	        IF (#new_packet) THEN
	            #_State := #STATE_INIT;
	        END_IF;
	        
	        
	END_CASE;
	
	EndAutomat:
	
	#CMD_CloseLodems := NOT #CMD_OpenLodems;
	
	// make new layer
	// 
	#make_gasket_layer := #s_lay_cmd_permission AND NOT #gaskets_busy AND (NOT (#mode_no_gasket OR #last_lay));
	
	
	
END_FUNCTION_BLOCK

FUNCTION "BoardDefinePosition" : Int
{ S7_Optimized_Access := 'FALSE' }
AUTHOR : Aspir
VERSION : 0.1
   VAR_INPUT 
      EnableRolling : Bool;   // нужна ли раскатка пакета
      PackL : Int;   // длина пакета с раскаткой
      PlankL : Int;   // длина доски
   END_VAR

   VAR CONSTANT 
      SafetyOffset : Int := 100;
   END_VAR


BEGIN
	IF (#EnableRolling) THEN
	    #BoardDefinePosition := #PackL;
	ELSIF (#PlankL = 0) THEN
	    #BoardDefinePosition := 6000;
	ELSE
	    #BoardDefinePosition := #PlankL + #SafetyOffset;
	END_IF;
END_FUNCTION

FUNCTION "SolveMovBoardPos" : Int
{ S7_Optimized_Access := 'FALSE' }
VERSION : 0.1
   VAR_INPUT 
      PlankLength : Int;
      Max_pos : Int;
      Min_pos : Int;
      Offset_chess : Int;
      PulseCount : Int;
   END_VAR

   VAR_TEMP 
      PlankLength_tmp : Int;
      Sub : Int;
      k : Real;
      b : Real;
   END_VAR


BEGIN
	IF (#PlankLength > #Max_pos) THEN
	    #PlankLength_tmp := #Max_pos;
	ELSIF (#PlankLength < #Min_pos) THEN
	    #PlankLength_tmp := #Min_pos;
	ELSE
	    #PlankLength_tmp := #PlankLength;
	END_IF;
	
	#Sub := (#Min_pos - #Max_pos);
	
	#k := INT_TO_REAL(#PulseCount) / #Sub;
	
	#b := - #Max_pos * #k;
	
	#SolveMovBoardPos := TRUNC_INT((#PlankLength_tmp + #Offset_chess)*#k + #b);
END_FUNCTION

FUNCTION_BLOCK "MovableBoard_CTRL"
{ S7_Optimized_Access := 'FALSE' }
VERSION : 0.1
   VAR_INPUT 
      BoardBase : Bool;   //   сигнал с дальнего концевика борта (знаем его позицию точно)
      ModeChanged : Bool;   //  был изменен режим
      Reset : Bool;   //   сбросить базу и позицию
      EncPos : Byte;   //   показания энкодера (код Грея)
      SetPos : Int;   //   абсолютное положение борта в импульсах
   END_VAR

   VAR_OUTPUT 
      CMD_Fwd : Bool;   //   команда на движение вперед
      CMD_Bwd : Bool;   //   команда на движение назад
      CMD_UP : Bool;   //   команда опустить борт
      CMD_DOWN : Bool;   //   команда поднять борт
      AutoMode : Bool;
      ResetVirtualPos : Bool;
      Position : Int;
   END_VAR

   VAR 
      DefinitionTag : Bool;   //   была определена позиция (база борта)
      ChangingPos : Bool;   //  в состоянии изменения позиции
      ShutUpAuto : Bool;   //  позицию изменил
      startOffset : Int;   //  начальный сдвиг
      curMicroPos : Int;
      curMicroPos_old : Int;
      curMacroPos : Int;
   END_VAR


BEGIN
	#ResetVirtualPos := FALSE;
	
	// условия для учета "перескоков" абсолютного энкодера на 256 позиций
	#curMicroPos := "Rev_G"(#EncPos);
	IF (#curMicroPos_old - #curMicroPos > 200) THEN
	    #curMacroPos := #curMacroPos + 1;
	END_IF;
	IF (#curMicroPos - #curMicroPos_old > 200) THEN
	    #curMacroPos := #curMacroPos - 1;
	END_IF;
	
	
	// Итоговое положение
	#Position := 256 * #curMacroPos + #curMicroPos - #startOffset;
	
	// Сброс базы
	IF #Reset THEN
	    #DefinitionTag := False;
	    #ChangingPos := FALSE;
	    #CMD_UP := FALSE;
	    #CMD_DOWN := FALSE;
	    
	    #ResetVirtualPos := TRUE;
	END_IF;
	
	// Доведем борт до концевика для уверенности в базе (нулевой точке)
	IF NOT #DefinitionTag THEN
	    #AutoMode := TRUE;
	    #CMD_UP := TRUE;
	    #CMD_DOWN := FALSE;
	    #CMD_Fwd := TRUE;
	    #CMD_Bwd := FALSE;
	    // Если дошли до дальнего концевика, знаем где мы, обнулим счетчик оборотов
	    IF (#BoardBase) THEN
	        #DefinitionTag := TRUE;
	        #ShutUpAuto := TRUE;
	        #curMacroPos := 0;
	        #startOffset := #curMicroPos;
	    END_IF;
	END_IF;
	
	
	IF (#ShutUpAuto) THEN
	    #AutoMode := False;
	    #ShutUpAuto := FALSE;
	END_IF;
	
	
	#ChangingPos := (#ChangingPos OR #ModeChanged);
	
	IF #ChangingPos AND #DefinitionTag THEN
	    #AutoMode := True;
	    #CMD_UP := True;
	    #CMD_DOWN := False;
	    
	    IF (ABS_INT(#Position - #SetPos) < 12) THEN
	        #ChangingPos := FALSE;
	        #ShutUpAuto := TRUE;
	        #CMD_UP := #SetPos < 30;
	        #CMD_DOWN := NOT #CMD_UP;
	        #CMD_Bwd := FALSE;
	        #CMD_Fwd := FALSE;
	        
	    ELSIF #Position > #SetPos THEN
	        #CMD_Bwd := FALSE;
	        #CMD_Fwd := TRUE;
	        
	    ELSE
	        #CMD_Bwd := TRUE;
	        #CMD_Fwd := FALSE;
	    END_IF;
	END_IF;
	
	
	#curMicroPos_old := #curMicroPos;
END_FUNCTION_BLOCK

FUNCTION "Rev_G" : Int
{ S7_Optimized_Access := 'FALSE' }
VERSION : 0.1
   VAR_INPUT 
      g_code : Byte;   // число (Код Грея)
   END_VAR

   VAR_TEMP 
      n : Byte;
   END_VAR


BEGIN
	#n := 0;
	
	WHILE NOT (#g_code = 0) DO
	    // Statement section WHILE
	    #n := #n XOR #g_code;
	    #g_code := SHR(IN := #g_code, N := 1);
	END_WHILE;
	
	#Rev_G := BYTE_TO_INT(#n);
END_FUNCTION

FUNCTION_BLOCK "FB_IM_PFM"
{ S7_Optimized_Access := 'FALSE' }
VERSION : 0.1
   VAR 
      M_233_Fork_PFM { S7_SetPoint := 'False'} : "FB_IM2x4";   // Вилы основной ПФМ
      M_232_Elevator_PFM : "FB_IM2x2S";   // Лифт основной ПФМ
      M_317_Carousel : "drive_CB_2x1";
      Elevator_brake_timer {InstructionName := 'TON'; LibVersion := '1.0'} : TON;
   END_VAR

   VAR_TEMP 
      Sert : Word;
   END_VAR


BEGIN
	
	REGION M_233
	    // Statement section REGION
	    #M_233_Fork_PFM(OnSig:="DGI".S15_2,
	                    OnSigLow:="DGI".S15_1,
	                    OffSig:= "DGI".S14_7,
	                    OffSigLow:="DGI".S15_0,
	                    sigFeedback:="DGI".F233K1 AND "DGI".K1_233U1,
	                    hasFeedback:=TRUE,
	                    Ready:="ALG".Ready_Sorting,
	                    Reset:="ALG".Reset OR "DGI".S76_2,
	                    btnAU:="ALG".Auto_Sorting OR "ServDB".M_233.BtnAU,
	                    btnDU:= NOT "ALG".Auto_Sorting AND "ServDB".M_233.BtnDU,
	                    prmDU:=TRUE,
	                    btnDU_ON:="ServDB".M_233.BtnFwd,
	                    btnDU_OF:= "ServDB".M_233.BtnBwd,
	                    btnDUStop:="ServDB".M_233.BtnCmdStop,
	                    btnMU:=NOT ("ALG".Auto_Sorting OR "ServDB".M_233.BtnDU),
	                    btnMU_ON:="DGI".S78_0,
	                    btnMU_OF:="DGI".E78_1,
	                    protection:=false,
	                    Set_T_notON:=T#20s,
	                    Set_T_notOFF:=T#20s,
	                    Set_T_notCMD:=T#500ms,
	                    Set_T_notFeedBack:=T#500ms,
	                    SpeedOn:=20,
	                    SpeedOnLow:=10,
	                    SpeedOff:=20,
	                    SpeedOffLow:=10,
	                    SpeedDU:="ServDB".M_233.SetSpeedDU,
	                    AU=>"ServDB".M_233.AU,
	                    DU=>"ServDB".M_233.DU,
	                    MU=>"ServDB".M_233.MU,
	                    Fault=>"ServDB".M_233.Fault,
	                    onOutFWD=>"ServDB".M_233.CMD_ON,
	                    onOutBWD=>"ServDB".M_233.CMD_OFF,
	                    PRM_btnDU_ON=>"ServDB".M_233.PrmBtnDU_ON,
	                    PRM_btnDU_OFF=>"ServDB".M_233.PrmBtnDU_OF
	                   
	    );
	    
	    
	    "K1-233X1" := "ALG".Ready_Sorting;
	    "K1-233U2" := #M_233_Fork_PFM.onOutFWD OR #M_233_Fork_PFM.onOutBWD;
	    "K1-233U2.2" := #M_233_Fork_PFM.onOutFWD;
	END_REGION
	
	REGION M_232
	    // Statement section REGION
	    #M_232_Elevator_PFM(onSig := "DGI".S16_2,
	                        offSig := "DGI".S16_1,
	                        sigFeedback := "DGI".F232K1 AND "DGI".K1_215U1,
	                        hasFeedback := true,
	                        btnUp := "ServDB".M_232.BtnFwd,
	                        btnDown := "ServDB".M_232.BtnBwd,
	                        btnStop := "ServDB".M_232.BtnCmdStop,
	                        Ready := "ALG".Ready_Sorting,
	                        Reset := "ALG".Reset OR "DGI".S76_2,
	                        prmDU := true,
	                        btnAU := "ServDB".M_232.BtnAU OR "ALG".Auto_Sorting,
	                        btnDU := "ServDB".M_232.BtnDU,
	                        btnMU := "DGI".E86_1 OR "DGI".E78_5 OR "DGI".S86_0 OR "DGI".S78_4 OR NOT ("ALG".Auto_Sorting OR "ServDB".M_232.BtnDU),
	                        btnMU_ON := "DGI".E86_1 OR "DGI".E78_5,
	                        btnMU_OF := "DGI".S86_0 OR "DGI".S78_4,
	                        set_time_notOn := T#1500ms,
	                        set_time_notOff := T#5000ms,
	                        set_time_notCMD := T#2000ms,
	                        setSpeedDU := "ServDB".M_232.SetSpeedDU,
	                        AU => "ServDB".M_232.AU,
	                        DU => "ServDB".M_232.DU,
	                        MU => "ServDB".M_232.MU,
	                        Fault => "ServDB".M_232.Fault,
	                        outFWD => "ServDB".M_232.CMD_ON,
	                        outBKD => "ServDB".M_232.CMD_OFF,
	                        setSpeed => "ServDB".M_317.SetSpeed
	    );
	    
	    "K1-232X1" := "ALG".Ready_Sorting;
	    // Управление тормозом
	    #Elevator_brake_timer(IN := #M_232_Elevator_PFM.outFWD XOR #M_232_Elevator_PFM.outBKD,
	                          PT := T#50ms
	    );
	    
	    "K1-232X1.1" := #Elevator_brake_timer.Q AND "DGI".K1_215U1;
	    
	    "K1-215U2.2" := #M_232_Elevator_PFM.outBKD;
	    "K1-215U2" := #M_232_Elevator_PFM.outFWD OR #M_232_Elevator_PFM.outBKD;
	END_REGION
	
	REGION M_317
	    
	    (* #M_317_Gasket_Carousel(OnSig:="DGI".F317K1 AND "DGI".K1_317U1,
	                           OnCom:= ("FB_Gasket_Carousel_DB".Carousel_FWD AND (NOT "B18.0")) OR "FB_Gasket_Carousel_DB".Carousel_BWD,
	                           Ready:="ALG".Ready_Sorting,
	                           Reset:="DGI".S76_2 OR "ALG".Reset,
	                           btnAU:= "ServDB".M_317.BtnAU OR "ALG".Auto_Sorting,
	                           btnDU:="ServDB".M_317.BtnDU,
	                           prmDU:=true,
	                           btnDU_ON:="ServDB".M_317.BtnFwd OR "ServDB".M_317.BtnBwd,
	                           btnDU_OF:= "ServDB".M_317.BtnCmdStop,
	                           btnMU:=NOT ("ServDB".M_317.BtnDU OR "ALG".Auto_Sorting) OR ("FB_Gasket_Carousel_DB".s_man_cntl AND "ALG".Auto_Sorting),
	                           btnMU_ON:="DGI".S84_1 OR "DGI".E84_2,
	                           btnMU_OF:= NOT ("DGI".S84_1 OR "DGI".E84_2),
	                           btn_Back_ON:= "ServDB".M_317.BtnBwd OR "DGI".E84_2 OR "FB_Gasket_Carousel_DB".Carousel_BWD,
	                           btn_Back_OFF:= NOT ("ServDB".M_317.BtnBwd OR "DGI".E84_2 OR "FB_Gasket_Carousel_DB".Carousel_BWD),
	                           Set_T_notON:=T#500ms,
	                           Set_T_notOFF:=T#500ms,
	                           setSpeedDU:="ServDB".M_317.SetSpeedDU,
	                           AU=>"ServDB".M_317.AU,
	                           DU=>"ServDB".M_317.DU,
	                           MU=>"ServDB".M_317.MU,
	                           BACK=>"ServDB".M_317.BACK,
	                           Alarm=>"ServDB".M_317.Alarm,
	                           Fault=>"ServDB".M_317.Fault,
	                           onOutFWD=>"ServDB".M_317.CMD_ON,
	                           onOutBWD=>"ServDB".M_317.CMD_OFF,
	                           PRM_btnDU_ON=>"ServDB".M_317.PrmBtnDU_ON,
	                           PRM_btnDU_OFF=>"ServDB".M_317.PrmBtnDU_OF,
	                           PRMbtn_Back_ON=>"ServDB".M_317.PRMbtn_Back_ON,
	                           PRMbtn_Back_OFF=>"ServDB".M_317.PRMbtn_Back_OFF,
	                           setSpeed=>"ServDB".M_317.SetSpeed
	    );
	    
	    
	    "K1-317X1" := "ALG".Ready_Sorting;
	    "K1-317U2" := #M_317_Gasket_Carousel.onOutFWD OR #M_317_Gasket_Carousel.onOutBWD;
	    "K1-317X1.1" := #M_317_Gasket_Carousel.onOutFWD OR #M_317_Gasket_Carousel.onOutBWD;
	    "K1-317U2.2" := #M_317_Gasket_Carousel.onOutBWD;
	    
	    *)
	    
	    #M_317_Carousel(i_ready := "ALG".Ready_Sorting,
	                    i_feedback := "DGI".F317K1 AND "DGI".K1_317U1,
	                    i_reset := "DGI".S76_2 OR "ALG".Reset,
	                    i_au_req := "ALG".Auto_Sorting,
	                    cmd_fwd := "FB_Gasket_Carousel_DB".Carousel_FWD AND NOT "B18.0",
	                    cmd_bwd := "FB_Gasket_Carousel_DB".Carousel_BWD,
	                    i_mu_req := ("FB_Gasket_Carousel_DB".s_man_cntl AND "ALG".Auto_Sorting) OR NOT ("ALG".Auto_Sorting OR "ServDB".M_317.BtnDU),
	                    mu_fwd := "DGI".S84_1,
	                    mu_bwd := "DGI".E84_2,
	                    i_du_req := "ServDB".M_317.BtnDU,
	                    du_fwd := "ServDB".M_317.BtnFwd,
	                    du_bwd := "ServDB".M_317.BtnBwd,
	                    i_speed_au := "FB_Gasket_Carousel_DB".Carousel_Speed,
	                    i_speed_mu_du := 7.0,
	                    ////////////////////////////////
	                    o_au => "ServDB".M_317.AU,
	                    o_du => "ServDB".M_317.DU,
	                    o_mu => "ServDB".M_317.MU,
	                    alarm => "ServDB".M_317.Alarm,
	                    o_fwd => "ServDB".M_317.CMD_ON,
	                    o_bwd => "ServDB".M_317.CMD_OFF);
	    
	    "K1-317X1" := "ALG".Ready_Sorting;
	    "K1-317U2" := #M_317_Carousel.o_fwd OR #M_317_Carousel.o_bwd;
	    "K1-317X1.1" := #M_317_Carousel.o_brake;
	    "K1-317U2.2" := #M_317_Carousel.o_bwd;
	    
	    #Sert := UNSCALE(IN := #M_317_Carousel.o_speed_vfd, HI_LIM := 50.0, LO_LIM := -50.0, BIPOLAR := TRUE, OUT => "K1-317U":P);
	    
	    
	    
	    
	END_REGION
END_FUNCTION_BLOCK

FUNCTION_BLOCK "FB_IM2x4"
{ S7_Optimized_Access := 'FALSE' }
AUTHOR : Ivanez
VERSION : 0.1
//Исполнительный механизм (2 команды, 4 положения - 2 конечных, 2 замедление)
   VAR_INPUT 
      OnSig : Bool;   //      Сигнал сработавшего открытого (выдвинутого)
      OnSigLow : Bool;   //      Сигнал сработавшего открытого (выдвинутого) замедление
      OffSig : Bool;   //      Сигнал сработавшего закрытого (задвинутого)
      OffSigLow : Bool;   //      Сигнал сработавшего закрытого (задвинутого) замедление
      OnCom : Bool;   //      Команда включения в автоматическом режиме
      OffCom : Bool;   //      Команда отключения в автоматическом режиме
      sigFeedback : Bool;   //      Обратная связь о том что устройство передвигается
      hasFeedback : Bool;   //      Флаг о наличии обратной связи по движению
      Ready : Bool;   //      Условие готовности
      Reset : Bool;   //      Сброс
      btnAU : Bool;   //      Перевести в Автоматическое управление
      btnDU : Bool;   //      Перевести в Дистанционное управление
      prmDU : Bool;   //      Разрешение на перевод в ДУ
      btnDU_ON : Bool;   //      Выдвинуть в дистанционном управлении
      btnDU_OF : Bool;   //      Задвинуть в дистанционном управлении
      btnDUStop : Bool;   //      Кнопка Останов
      btnMU : Bool;   //      Перевести в местное управление
      btnMU_ON : Bool;   //      Включить в местном управлении
      btnMU_OF : Bool;   //      Отключить в местном управлении
      protection : Bool;   //      Условие включение защиты
      Set_T_notON : Time;   //      Задержа на формирование неоткрытия
      Set_T_notOFF : Time;   //      Задержа на формирование незакрытия
      Set_T_notCMD : Time;   //      Задержа на формирование отсутсвия команды
      Set_T_notFeedBack : Time;   // Задержка на формирование ошибки отсутствия обратной связи
      SpeedOn : Real;   //     Задание на скорость выдвижения
      SpeedOnLow : Real;   //     Задание на скорость выдвижения низкая
      SpeedOff : Real;   //     Задание на скорость задвижения
      SpeedOffLow : Real;   //     Задание на скорость задвижения низкая
      SpeedDU : Real;   //     Задание на скорость в ДУ
   END_VAR

   VAR_OUTPUT 
      AU : Bool;   //      Автоматическое управление (АУ)
      DU : Bool;   //      Дистанционное управление (ДУ)
      MU : Bool;   //      Местное управление (МУ)
      notON : Bool;   //      Предупреждение о невключении
      notOFF : Bool;   //      Предупреждение о неотключении
      notCMD : Bool;   //      Предупреждение об отсутствие команды
      notFeedBack : Bool;   // Предупреждение об отсутствии обратной связи
      Fault : Bool;   //      Неисправность
      onOutFWD : Bool;   //      Сигнал на открытие (выдвинуть)
      onOutBWD : Bool;   //      Сигнал на закрытие (задвинуть)
      PRM_btnDU_ON : Bool;   //      Разрешение кнопки включения в ДУ
      PRM_btnDU_OFF : Bool;   //      Разрешение кнопки отключения в ДУ
      SetSpeed : Real;   //     Задание на ПЧ
   END_VAR

   VAR 
      speedLow_forward : Bool;
      speedLow_revers : Bool;
      checker_forward : Bool;
      checker_revers : Bool;
      unkn_state : Bool;   //     Неизвестное состояние
      wrong_state : Bool;   //     Некорректное состояние
      sigOnOut : Bool;   //      Сигналоткрытия
      sigOffOut : Bool;   //      Сигнал закрытия
      T_notON_TON {InstructionName := 'TON'; LibVersion := '1.0'; S7_SetPoint := 'False'} : TON;   //      Таймер неоткрытия
      T_notOFF_TON {InstructionName := 'TON'; LibVersion := '1.0'; S7_SetPoint := 'False'} : TON;   //      Таймер незакрытия
      T_notCMD_TON {InstructionName := 'TON'; LibVersion := '1.0'; S7_SetPoint := 'False'} : TON;   //      Таймер отстутствия
      T_notFeedBack_TON {InstructionName := 'TON'; LibVersion := '1.0'} : TON;   // Таймер отсутствия обратной связи
   END_VAR


BEGIN
	
	//Формирование автоматического управления
	IF #btnAU THEN
	    #AU := true;
	    #DU := false;
	    #MU := false;
	END_IF;
	//Формирование дистанционного управления 
	IF #btnDU THEN
	    #DU := true;
	    #AU := false;
	    #MU := false;
	END_IF;
	//Формирование местного управления
	IF #btnMU THEN
	    #MU := true;
	    #AU := false;
	    #DU := false;
	END_IF;
	
	IF NOT #AU AND NOT #DU AND NOT #MU THEN
	    #MU := true;
	END_IF;
	
	//Разрешения кнопок управления
	#PRM_btnDU_ON := (NOT #OnSig AND #DU OR #notON);
	#PRM_btnDU_OFF := (NOT #OffSig AND #DU OR #notOFF);
	
	
	// Контроль скорости
	// 
	// триггеры замедления
	// 
	#speedLow_forward := (#speedLow_forward OR #OnSigLow AND #sigOnOut) AND NOT (#OnSig OR #OnSigLow AND #sigOffOut);
	#speedLow_revers := (#speedLow_revers OR #OffSigLow AND #sigOffOut) AND NOT (#OffSig OR #OffSigLow AND #sigOnOut);
	#checker_forward := (#checker_forward OR #OffSig) AND NOT #OffSigLow;
	#checker_revers := (#checker_revers OR #OnSig) AND NOT #OnSigLow;
	
	IF (#sigOnOut) THEN
	    IF (#speedLow_forward OR #checker_revers) THEN
	        #SetSpeed := #SpeedOnLow;
	    ELSE
	        #SetSpeed := #SpeedOn;
	    END_IF;
	    
	    
	ELSIF (#sigOffOut) THEN
	    IF (#speedLow_revers OR #checker_forward) THEN
	        #SetSpeed := #SpeedOffLow;
	    ELSE
	        #SetSpeed := #SpeedOff;
	    END_IF;
	ELSE
	    #SetSpeed := 0;
	END_IF;
	
	//------------------------------------------------
	//Формирование выходного сигнала открытия (выдвижение)
	#sigOnOut := #Ready AND ((#sigOnOut
	OR #AU AND #OnCom
	OR #DU AND #btnDU_ON
	OR #MU AND #btnMU_ON)
	AND NOT (#OnSig
	OR #AU AND ( #OffCom)
	OR #DU AND (#btnDU_OF OR #btnDUStop)
	OR #MU AND (NOT #btnMU_ON OR #btnMU_OF)
	OR #notON
	OR #wrong_state
	));
	
	//Формирование выходного сигнала закрытия (задвижение)
	#sigOffOut := #Ready AND ((#sigOffOut
	OR #AU AND #OffCom
	OR #DU AND #btnDU_OF
	OR #MU AND #btnMU_OF)
	AND NOT (#OffSig
	OR #AU AND (#OnCom)
	OR #DU AND (#btnDU_ON OR #btnDUStop)
	OR #MU AND (#btnMU_ON OR NOT #btnMU_OF)
	OR #notOFF
	OR #wrong_state
	));
	
	//Выбор выхода 
	#onOutFWD := #sigOnOut;
	#onOutBWD := #sigOffOut;
	
	
	//Неизвестное состояние
	#unkn_state := NOT (#OnSig OR #OffSig OR #onOutBWD OR #onOutFWD) AND NOT #Reset;
	
	//Некорректное состояние
	#wrong_state := (#wrong_state
	OR #OnSig AND #OffSig
	OR #OnSig AND #OffSigLow
	OR #OnSigLow AND #OffSigLow
	OR #OnSigLow AND #OffSig
	) AND NOT #Reset;
	
	
	#T_notON_TON(
	             IN := ( #sigOnOut AND NOT #sigOffOut AND NOT #OnSig AND NOT #Reset ),
	             PT := #Set_T_notON
	);
	
	#notON := (#notON OR #T_notON_TON.Q) AND NOT #Reset;
	
	#T_notCMD_TON(
	              IN := ( NOT #sigOnOut AND NOT #sigOffOut AND (#sigFeedback AND #hasFeedback) AND NOT #Reset),
	              PT := #Set_T_notCMD
	);
	
	#notCMD := (#notCMD OR #T_notCMD_TON.Q) AND NOT #Reset;
	
	
	#T_notOFF_TON(
	              IN := (NOT #sigOnOut AND #sigOffOut AND NOT #OffSig AND NOT #Reset),
	              PT := #Set_T_notOFF
	);
	
	#notOFF := (#notOFF OR #T_notOFF_TON.Q) AND NOT #Reset;
	
	#T_notFeedBack_TON(
	                   IN := (#sigOnOut OR #sigOffOut) AND NOT (#sigFeedback AND #hasFeedback) AND NOT #Reset,
	                   PT := #Set_T_notFeedBack
	);
	
	#notFeedBack := (#notFeedBack OR #T_notFeedBack_TON.Q) AND NOT #Reset;
	
	//Обобщенная неисправность
	#Fault := #notON OR #notOFF OR #notCMD OR #notFeedBack OR #wrong_state OR #unkn_state;
END_FUNCTION_BLOCK

FUNCTION_BLOCK "FB_IM2x2S"
{ S7_Optimized_Access := 'FALSE' }
VERSION : 0.1
//------------------------------------------------------------------------------------
//  Declaration of Variables
//------------------------------------------------------------------------------------
   VAR_INPUT 
      onSig : Bool;   //      Сигнал верхнего концевика
      offSig : Bool;   //      Сигнал нижнего концевика
      sigFeedback : Bool;   //      Обратная связь о том что устройство передвигается
      hasFeedback : Bool;   //      Флаг о наличии обратной связи по движению
      comUp : Bool;   //      Команда на подъем оборудования в автомате
      comDown : Bool;   //      Команда на спуск оборудования в автомате
      btnUp : Bool;   //      Кнопка на подъем лифта
      btnDown : Bool;   //      Кнопка на спуск лифта
      btnStop : Bool;   //      Кнопка Останов
      Ready : Bool;   //      Условие готовности
      Reset : Bool;   //      Сброс
      prmDU : Bool;   //      Разрешение на перевод в ДУ
      btnAU : Bool;   //      Команда на перевод в АУ
      btnDU : Bool;   //      Команда на пеервод в ДУ
      btnMU : Bool;
      btnMU_ON : Bool;   //      Включить в местном управлении
      btnMU_OF : Bool;   //      Отключить в местном управлении
      set_time_notOn : Time;   //      установка времени на неВКЛючение
      set_time_notOff : Time;   //      установка времени на неВЫКЛючение
      set_time_notCMD : Time;   //      установка времени отсутсивие команды
      setSpeedAU : Real;   //      Скорость в режиме автомат
      setSpeedDU : Real;   //      Скорость в режиме ДУoutputs
   END_VAR

   VAR_OUTPUT 
      AU : Bool;   //      Режим - Автомат
      DU : Bool;   //      Режим - ДистанционноеAlarm : Bool; // Авария
      MU : Bool;
      Fault : Bool;   //      Неисправность
      outFWD : Bool;   //      Сигнал о движении вверх (вперед)
      outBKD : Bool;   //      Сигнал о движении вниз (назад)
      notOn : Bool;   //      Сигнал на неВКЛючение
      notCMD : Bool;   //      Отсутствие команды
      notOff : Bool;   //      Сигнал на неВЫКЛючение
      wrong_state : Bool;   //      Некорректное состояние
      wrong_CMD : Bool;   // неверная команда
      setSpeed : Real;   //      скорость в автомате для частотникаvariables
   END_VAR

   VAR 
      timer_notOn {InstructionName := 'TON'; LibVersion := '1.0'} : TON;
      timer_notOff {InstructionName := 'TON'; LibVersion := '1.0'} : TON;
      timer_notCMD {InstructionName := 'TON'; LibVersion := '1.0'} : TON;
   END_VAR


BEGIN
	//Формирование автоматического управления
	IF #btnAU THEN
	    #AU := true;
	    #DU := false;
	    #MU := false;
	END_IF;
	//Формирование дистанционного управления 
	IF #btnDU THEN
	    #DU := true;
	    #AU := false;
	    #MU := false;
	END_IF;
	//Формирование местного управления
	IF #btnMU THEN
	    #MU := true;
	    #AU := false;
	    #DU := false;
	END_IF;
	
	IF NOT #AU AND NOT #DU AND NOT #MU THEN
	    #MU := true;
	END_IF;
	
	#outFWD := #Ready
	AND ((#outFWD
	OR #DU AND #btnUp
	OR #MU AND #btnMU_ON
	OR #AU AND #comUp)
	AND NOT (#Fault OR #onSig OR (#DU AND #btnStop) OR (#AU AND NOT #comUp) OR (#MU AND NOT #btnMU_ON))
	);
	
	#outBKD := #Ready
	AND ((#outBKD
	OR #DU AND #btnDown
	OR #MU AND #btnMU_OF
	OR #AU AND #comDown)
	AND NOT (#Fault OR #offSig OR (#DU AND #btnStop) OR (#AU AND NOT #comDown) OR (#MU AND NOT #btnMU_OF))
	);
	
	#timer_notOn(IN := (NOT #outBKD AND #outFWD) AND NOT (#sigFeedback AND #hasFeedback) AND NOT #Reset,
	             PT := #set_time_notOn);
	#notOn := (#notOn OR #timer_notOn.Q) AND NOT #Reset;
	
	// Не едет наверх
	// Проверка на отсутствие команд
	#timer_notCMD(IN := NOT (#outBKD OR #outFWD) AND (#sigFeedback AND #hasFeedback) AND NOT #Reset,
	              PT := #set_time_notCMD);
	#notCMD := (#notCMD OR #timer_notCMD.Q) AND NOT #Reset;
	
	// Не едет вниз
	#timer_notOff(IN := (#outBKD AND NOT #outFWD) AND NOT (#sigFeedback AND #hasFeedback) AND NOT #Reset,
	              PT := #set_time_notOff);
	#notOff := (#notOff OR #timer_notOff.Q) AND NOT #Reset;
	
	#wrong_CMD := (#wrong_CMD OR (#outFWD AND #outBKD)) AND NOT #Reset;
	
	#wrong_state := #onSig AND #offSig;
	
	#Fault := #notOn OR #notOff OR #notCMD OR #wrong_state OR #wrong_CMD;
	
	IF #DU THEN
	    #setSpeed := #setSpeedDU;
	ELSE
	    #setSpeed := #setSpeedAU;
	END_IF;
	
	
END_FUNCTION_BLOCK

FUNCTION_BLOCK "FB_HydroStations"
{ S7_Optimized_Access := 'FALSE' }
VERSION : 0.1
   VAR 
      Upor_resetter { S7_SetPoint := 'False'} : "CyclicSignal";
      Movable_side_resetter : "CyclicSignal";
      Gasket_Ramp_sync : "CyclicSignal";
      DefectDrop_resetter : "CyclicSignal";
      Board_Rotator { S7_SetPoint := 'False'} : "FB_IM2x0";   // переворот доски
      Defect_Drop : "FB_IM2x0";   // сброс в брак
      Upor_Sorting { S7_SetPoint := 'False'} : "FB_IM2x0";   // упор перед зоной оценки (поштучки)
      Upor_Defective : "FB_IM2x2";   // упоры ПФМ брака
      Gasket_Supplier { S7_SetPoint := 'False'} : "FB_IM2x0";   // выдача прокладки на карусель
      Gasket_Ramp : "FB_IM2x3";   // рама прокладок
      Gasket_Lodems : "FB_IM2x2";   // Стакан прокладок на раме
      Forks_Pitcher : "FB_IM2x2";   // подъемник вил ПФМ
      Movable_Side : "FB_IM2x0";   // Подвижный борт
      Upor_PFM : "FB_IM2x0";   // упоры перед пощштучной выдачей
      M_221_Large_HydroStationDrive : "FB_HySt_Drive_PassValve";   // двигатель маленькой гидростанции
      M_337_Small_HydroStationDrive : "FB_HySt_Drive_PassValve";   // двигатель большой гидростанции
   END_VAR


BEGIN
	REGION Small_HydroStationMechs
	    // Statement section REGION
	    
	    #Board_Rotator(Ready:="ALG".Ready_Sorting AND #M_337_Small_HydroStationDrive.CMD_DriveOn,
	                   Reset:="ALG".Reset,
	                   btnMU := TRUE,
	                   btnMU_On:="DGI".S88_7,
	                   btnMU_Off:=NOT "DGI".S88_7,
	                   set_T_On:=T#1s,
	                   set_T_Off:=T#1s,
	                   outFwd=> "Y223_1",
	                   outBwd=>"Y223_2"
	    );
	    
	    #DefectDrop_resetter(count:=240,
	                         Meandr_counter:="ALG".Meandr);
	    
	    #Defect_Drop(
	                 Ready:="ALG".Ready_Sorting AND #M_337_Small_HydroStationDrive.CMD_DriveOn,
	                 Reset:="ALG".Reset OR #DefectDrop_resetter.change,
	                 btnAU:= "ALG".Auto_Sorting,
	                 set_T_On:=T#2s,
	                 set_T_Off:=T#2200ms,
	                 outFwd => "Y223_4",
	                 outBwd => "Y223_3"
	    );
	    
	    #Upor_Sorting(Ready := "ALG".Ready_Sorting  AND #M_337_Small_HydroStationDrive.CMD_DriveOn,
	                  Reset := "ALG".Reset,
	                  btnAU := "ALG".Auto_Sorting,
	                  btnMU:=NOT ("ALG".Auto_Sorting),
	                  btnMU_On:= "DGI".S80_0,
	                  btnMU_Off:= "DGI".E80_1,
	                  set_T_On := T#1s,
	                  set_T_Off := T#500ms,
	                  outFwd => "Y323_2",
	                  outBwd => "Y323_1"
	    );
	    
	    #Upor_Defective(OnSig:="DGI".FC_23_6,
	                    OffSig:="DGI".FC_23_7,
	                    Ready:="ALG".Ready_defect AND #M_337_Small_HydroStationDrive.CMD_DriveOn,
	                    Reset:="ALG".Reset OR "DGI".S76_2,
	                    btnAU:="ALG".Auto_defect,
	                    btnMU:="DGI".S90_6 OR "DGI".E90_7, // OR "DGI".S80_0 OR "DGI".E80_1,
	                    btnMU_ON:= "DGI".S90_6,
	                    btnMU_OF:="DGI".E90_7,
	                    Set_T_notON:=T#7s,
	                    Set_T_notOFF:=T#7s,
	                    onOutFWD=>"Upor_brak_up",
	                    onOutBWD=>"Upor_brak_down"
	                    
	    );
	    
	END_REGION
	
	REGION Large_HydroStationMechs
	    // Statement section REGION
	    // 
	
	    #Gasket_Supplier(Ready := "ALG".Ready_Sorting AND #M_221_Large_HydroStationDrive.CMD_DriveOn,
	                     Reset := "ALG".Reset OR "DGI".S76_2,
	                     btnAU := "ALG".Auto_Sorting,
	                     btnDU:="ServDB".GasketSupplier.BtnDU,
	                     btnMU:=NOT ("ALG".Auto_Sorting OR "ServDB".GasketSupplier.BtnDU),
	                     btnDU_On:="ServDB".GasketSupplier.BtnFwd,
	                     btnDU_Off:="ServDB".GasketSupplier.BtnBwd,
	                     set_T_On := T#1s,
	                     set_T_Off := T#700ms,
	                     AU=>"ServDB".GasketSupplier.AU,
	                     DU=>"ServDB".GasketSupplier.DU,
	                     MU=>"ServDB".GasketSupplier.MU,
	                     outFwd => "Line4_2",
	                     outBwd => "Line4_1"
	    );
	    
	    #Gasket_Ramp_sync(count:=100,
	                      Meandr_counter:="ALG".Meandr);
	    
	    
	    #Gasket_Ramp(upSig:="DGI".B18_0,
	                 midSig:="DGI".S18_2,
	                 dnSig:="DGI".GasketRampSqueeze_timer.Q,
	                 Ready:="ALG".Ready_Sorting AND #M_221_Large_HydroStationDrive.CMD_DriveOn,
	                 Reset:="ALG".Reset OR "DGI".S76_2,
	                 btnAU:="ALG".Auto_Sorting OR "ALG".VirtualAuto,
	                 btnMU:= NOT ("ALG".Auto_Sorting OR "ALG".VirtualAuto),
	                 btnMU_ON:="DGI".E84_6 OR "DGI".S78_6,
	                 btnMU_OF:="DGI".S84_5 OR "DGI".E78_7,
	                 sync_sig:=#Gasket_Ramp_sync.change OR "ALG".RampSyncSig,
	                 set_time_notRun:=T#10s,
	                 outUp=>"Line5_2",
	                 outDn=>"Line5_1"
	    );
	   
	    
	    #Gasket_Lodems(OnSig := "DGI".B18_4,
	                   OffSig := "DGI".B18_5,
	                   Ready := "ALG".Ready_Sorting AND #M_221_Large_HydroStationDrive.CMD_DriveOn,
	                   Reset := "ALG".Reset OR "DGI".S76_2,
	                   btnAU := "ALG".Auto_Sorting,
	                   btnMU := NOT "ALG".Auto_Sorting,
	                   btnMU_ON := "DGI".S84_7,
	                   btnMU_OF := "DGI".E85_0,
	                   Set_T_notON := T#2s,
	                   Set_T_notOFF := T#2s,
	                   onOutFWD => "Line6_2",
	                   onOutBWD => "Line6_1"
	                   
	    );
	    
	    #Movable_side_resetter(count:=500,
	                           Meandr_counter:="ALG".Meandr);
	    
	    #Movable_Side(Ready := "ALG".Ready_Sorting AND #M_221_Large_HydroStationDrive.CMD_DriveOn,
	                  Reset := "ALG".Reset OR #Movable_side_resetter.change OR "MovableBoard_CTRL_DB".ResetVirtualPos,
	                  btnAU := "MovableBoard_CTRL_DB".AutoMode,
	                  btnMU:=NOT "MovableBoard_CTRL_DB".AutoMode,
	                  btnMU_On:="DGI".btn_Cnrl_Mov_Side.CMD_ON,
	                  btnMU_Off:="DGI".btn_Cnrl_Mov_Side.CMD_OFF,
	                  set_T_On := T#700ms,
	                  set_T_Off := T#700ms,
	                  outFwd => "Line3_2",
	                  outBwd => "Line3_1"
	                  
	    );
	    
	    #Forks_Pitcher(OnSig:= false,//"DGI".B15_7,
	                   OffSig:= "DGI".B15_5,
	                   Ready:="ALG".Ready_Sorting AND #M_221_Large_HydroStationDrive.CMD_DriveOn,
	                   Reset:="ALG".Reset OR "DGI".S76_2,
	                   btnAU:="ALG".Auto_Sorting,
	                   prmDU:=true,
	                   btnMU:=NOT "ALG".Auto_Sorting,
	                   btnMU_ON:= "DGI".S78_2,
	                   btnMU_OF:= "DGI".E78_3,
	                   Set_T_notON:=T#20m,
	                   Set_T_notOFF:=T#2s,
	                   onOutFWD=>"Line1_2",
	                   onOutBWD=>"Line1_1"
	    );
	    
	    #Upor_resetter(count:=90,
	                   Meandr_counter:="ALG".Meandr);
	    
	    #Upor_PFM(Ready := "ALG".Ready_Sorting AND #M_221_Large_HydroStationDrive.CMD_DriveOn,
	              Reset := "ALG".Reset OR "DGI".btn_ResetUporLine.CMD_ON OR #Upor_resetter.change,
	              btnAU := "ALG".Auto_Sorting,
	              set_T_On := "ALG".SqueezeUporPFM,// T#20m,
	              set_T_Off := T#120ms,
	              outFwd => "Line2_1",
	              outBwd => "Line2_2"
	    );
	    
	END_REGION
	
	#M_221_Large_HydroStationDrive(OnSig:="DGI".F221K1,
	                               Ready:="ALG".Ready_Sorting,
	                               Reset:="DGI".S76_2 OR "ALG".Reset ,
	                               sigValveFault:=("Line1_1" AND "Line1_2") OR
	                               ("Line2_1" AND "Line2_2") OR
	                               ("Line3_1" AND "Line3_2") OR
	                               ("Line4_1" AND "Line4_2") OR
	                               ("Line5_1" AND "Line5_2") OR
	                               ("Line6_1" AND "Line6_2"),
	                               
	                               PerepuskOn:=("Line1_1" OR "Line1_2") OR
	                               #Upor_PFM.inWork OR
	                               #Movable_Side.inWork OR
	                               #Gasket_Supplier.inWork OR
	                               ("Line5_1" OR "Line5_2") OR
	                               ("Line6_1" OR "Line6_2"),
	                                
	                               Set_T_notOn:=T#500ms,
	                               Set_T_notOFF:=T#500ms,
	                               CMD_DriveOn=>"K1-221X1",
	                              CMD_PassValveOn=>"Perepusk"
	);
	
	#M_337_Small_HydroStationDrive(OnSig:="DGI".F337K1,
	                               Ready:="ALG".Ready_Sorting,
	                               Reset:="DGI".S76_2 OR "ALG".Reset,
	                               sigValveFault:= ("Y223_1" AND "Y223_2") OR ("Y223_3" AND "Y223_4") OR ("Y323_1"
	                               AND "Y323_2") OR ("Upor_brak_up" AND "Upor_brak_down"),
	                               PerepuskOn:=("Y223_1" OR "Y223_2") OR ("Y223_3" OR "Y223_4") OR ("Y323_1"
	                               OR "Y323_2") OR ("Upor_brak_up" OR "Upor_brak_down"),
	                               Set_T_notOn:=T#500ms,
	                               Set_T_notOFF:=T#500ms,
	                               CMD_DriveOn=>"K1-337K1",
	                               CMD_PassValveOn=>"Y223.3"
	);
	
	
END_FUNCTION_BLOCK

FUNCTION_BLOCK "CyclicSignal"
{ S7_Optimized_Access := 'FALSE' }
VERSION : 0.1
   VAR_INPUT 
      count : Int;   // количество полусекунд
      Meandr_counter : Int;   // счетчик меандра
   END_VAR

   VAR_OUTPUT 
      meandr : Bool;
      change : Bool;
   END_VAR

   VAR 
      trig_cycled : Bool;
      Memento_counter : Int;
   END_VAR

   VAR_TEMP 
      on_cond : Bool;
   END_VAR


BEGIN
	#on_cond := #Meandr_counter MOD #count = 0;
	
	#change := FALSE;
	
	IF (#on_cond AND NOT #trig_cycled) THEN
	    #change := TRUE;
	    #meandr := NOT #meandr;
	    #Memento_counter := #Meandr_counter;
	END_IF;
	
	#trig_cycled := (#trig_cycled OR #on_cond) AND (#Meandr_counter = #Memento_counter);
END_FUNCTION_BLOCK

FUNCTION_BLOCK "FB_IM2x0"
{ S7_Optimized_Access := 'FALSE' }
VERSION : 0.1
   VAR_INPUT 
      OnCom : Bool;   // команда вперед/вверх в авто
      OffCom : Bool;   // команда назад/вниз авто
      Ready : Bool;   // готовность
      Reset : Bool;   // сброс ошибки
      btnAU : Bool;   // авто режим 
      btnDU : Bool;   // режим ДУ
      btnMU : Bool;   // местное управление
      btnDU_On : Bool;   // вперед/вверх ДУ
      btnDU_Off : Bool;   // назад/вниз ДУ
      btnMU_On : Bool;   // вперед/вверх МУ
      btnMU_Off : Bool;   // назад/вниз МУ
      set_T_On : Time;   // время на сработку механизма вверх
      set_T_Off : Time;   // время на сработку механизма вниз
   END_VAR

   VAR_OUTPUT 
      AU : Bool;
      DU : Bool;
      MU : Bool;
      outFwd : Bool;   // сигнал вперед/вниз
      outBwd : Bool;   // сигнал назад/вниз
      inWork : Bool;   // сигнал в работе
   END_VAR

   VAR 
      virtualOnSig : Bool;   // виртуальный верхний конфевик
      virtualOffSig : Bool;   // виртуальный нижний концевик
      timer_full_On {InstructionName := 'TON'; LibVersion := '1.0'} : TON;
      timer_full_Off {InstructionName := 'TON'; LibVersion := '1.0'; S7_SetPoint := 'False'} : TON;
   END_VAR


BEGIN
	//Формирование автоматического управления
	IF #btnAU THEN
	    #AU := true;
	    #DU := false;
	    #MU := false;
	END_IF;
	//Формирование дистанционного управления 
	IF #btnDU THEN
	    #DU := true;
	    #AU := false;
	    #MU := false;
	END_IF;
	//Формирование местного управления
	IF #btnMU THEN
	    #MU := true;
	    #AU := false;
	    #DU := false;
	END_IF;
	
	IF NOT #AU AND NOT #DU AND NOT #MU THEN
	    #MU := true;
	END_IF;
	
	#outFwd := #Ready AND ((#outFwd 
	OR #AU AND #OnCom
	OR #DU AND #btnDU_On
	OR #MU AND #btnMU_On)
	AND NOT (
	#virtualOnSig
	OR #AU AND #OffCom
	OR #DU AND #btnDU_Off
	OR #MU AND #btnMU_Off
	));
	
	#outBwd := #Ready AND (( #outBwd
	OR #AU AND #OffCom
	OR #DU AND #btnDU_Off
	OR #MU AND #btnMU_Off
	)
	AND NOT
	(#virtualOffSig
	OR #AU AND #OnCom
	OR #DU AND #btnDU_On
	OR #MU AND #btnMU_On));
	
	#timer_full_On(IN:=#outFwd AND NOT #Reset,
	               PT:=#set_T_On
	);
	
	#virtualOnSig := (#virtualOnSig OR #timer_full_On.Q) AND NOT #outBwd AND NOT #Reset;
	
	#timer_full_Off(IN:=#outBwd AND NOT #Reset,
	                PT:=#set_T_Off
	);
	
	#virtualOffSig := (#virtualOffSig OR #timer_full_Off.Q) AND NOT #outFwd  AND NOT #Reset;
	
	#inWork := #outBwd XOR #outFwd;
END_FUNCTION_BLOCK

FUNCTION_BLOCK "FB_IM2x2"
{ S7_Optimized_Access := 'FALSE' }
AUTHOR : Ivanez
VERSION : 0.1
//Исполнительный механизм (2 команды, 2 положения)
   VAR_INPUT 
      OnSig : Bool;   //      Сигнал сработавшего открытого (выдвинутого)
      OffSig : Bool;   //      Сигнал сработавшего закрытого (задвинутого)
      sigFeedBack : Bool;   // Обратная связь
      hasFeedBack : Bool;   // Есть ли обратная связь
      OnCom : Bool;   //      Команда включения в автоматическом режиме
      OffCom : Bool;   //      Команда отключения в автоматическом режиме
      Ready : Bool;   //      Условие готовности
      Reset : Bool;   //      Сброс
      btnAU : Bool;   //      Перевести в Автоматическое управление
      btnDU : Bool;   //      Перевести в Дистанционное управление
      prmDU : Bool;   //      Разрешение на перевод в ДУ
      btnDU_ON : Bool;   //      Включить в дистанционном управлении
      btnDU_OF : Bool;   //      Отключить в дистанционном управлении
      btnMU : Bool;   //      Перевести в местное управление
      btnMU_ON : Bool;   //      Включить в местном управлении
      btnMU_OF : Bool;   //      Отключить в местном управлении
      protection : Bool;   //      Условие включение защиты
      Set_T_notON : Time;   //      Задержа на формирование неоткрытие
      Set_T_notOFF : Time;   //      Задержа на формирование незакрытие
      time_notFeedBack : Time;
      time_notCMD : Time;
      setSpeedAU : Real;   //      Скорость в режиме автомат
      setSpeedDU : Real;   //      Скорость в режиме ДУoutputs
   END_VAR

   VAR_OUTPUT 
      AU : Bool;   //      Автоматическое управление (АУ)
      DU : Bool;   //      Дистанционное управление (ДУ)
      MU : Bool;   //      Местное управление (МУ)
      wrong_state : Bool;   //  Некорректное состояние
      notON : Bool;   //      Предупреждение о невключении
      notOFF : Bool;   //      Предупреждение о неотключении
      notCMD : Bool;
      notFeedBack : Bool;
      Fault : Bool;   //      Неисправность
      onOutFWD : Bool;   //      Сигнал на открытие (выдвинуть)
      onOutBWD : Bool;   //      Сигнал на закрытие (задвинуть)
      PRM_btnDU_ON : Bool;   //      Разрешение кнопки включения в ДУ
      PRM_btnDU_OFF : Bool;   //      Разрешение кнопки отключения в ДУ
      setSpeed : Real;   //      скорость в автомате для частотникаvariables
   END_VAR

   VAR 
      sigOnOut : Bool;   //      Сигналоткрытия
      sigOffOut : Bool;   //      Сигнал закрытия
      T_notON_TON {InstructionName := 'TON'; LibVersion := '1.0'; S7_SetPoint := 'False'} : TON;   //      Таймер неоткрытия
      T_notOFF_TON {InstructionName := 'TON'; LibVersion := '1.0'; S7_SetPoint := 'False'} : TON;   //      Таймер незакрытия
      T_notFeedback {InstructionName := 'TON'; LibVersion := '1.0'; S7_SetPoint := 'False'} : TON;
      T_notCMD {InstructionName := 'TON'; LibVersion := '1.0'; S7_SetPoint := 'False'} : TON;
   END_VAR


BEGIN
	//Формирование автоматического управления
	IF #btnAU THEN
	    #AU := true;
	    #DU := false;
	    #MU := false;
	END_IF;
	//Формирование дистанционного управления 
	IF #btnDU THEN
	    #DU := true;
	    #AU := false;
	    #MU := false;
	END_IF;
	//Формирование местного управления
	IF #btnMU THEN
	    #MU := true;
	    #AU := false;
	    #DU := false;
	END_IF;
	
	IF NOT #AU AND NOT #DU AND NOT #MU THEN
	    #MU := true;
	END_IF;
	
	//Разрешения кнопок управления
	#PRM_btnDU_ON := (NOT #OnSig AND #DU OR #notON);
	#PRM_btnDU_OFF := (NOT #OffSig AND #DU OR #notOFF);
	
	//Формирование выходного сигнала открытия (выдвижение)
	#sigOnOut := #Ready AND ((#sigOnOut
	OR #AU AND #OnCom
	OR #DU AND #btnDU_ON
	OR #MU AND #btnMU_ON
	)
	AND NOT
	(#OnSig
	OR #AU AND #OffCom
	OR #DU AND #btnDU_OF
	OR #MU AND #btnMU_OF
	OR #Fault));
	
	
	//Формирование выходного сигнала закрытия (задвижение)
	#sigOffOut := #Ready AND ((#sigOffOut
	OR #AU AND #OffCom
	OR #DU AND #btnDU_OF
	OR #MU AND #btnMU_OF
	)
	AND NOT
	(#OffSig
	OR #AU AND #OnCom
	OR #DU AND #btnDU_ON
	OR #MU AND #btnMU_ON
	OR #Fault));
	
	//Выбор выхода ВПЕРЕД НАЗАД
	#onOutFWD := #sigOnOut;
	#onOutBWD := #sigOffOut;
	
	//Неисправности
	#T_notON_TON(
	             IN := (#sigOnOut AND NOT #OnSig AND NOT #Reset),
	             PT := #Set_T_notON
	);
	
	#notON := (#notON OR #T_notON_TON.Q) AND NOT #Reset;
	
	#T_notOFF_TON(
	              IN := (#sigOffOut AND NOT #OffSig AND NOT #Reset),
	              PT := #Set_T_notOFF
	);
	
	#notOFF := (#notOFF OR #T_notOFF_TON.Q) AND NOT #Reset;
	
	
	#T_notFeedback(
	               IN := ((#sigOffOut OR #sigOnOut) AND NOT #sigFeedBack AND #hasFeedBack AND NOT #Reset),
	               PT := #time_notFeedBack
	);
	
	#notFeedBack := (#notFeedBack OR #T_notFeedback.Q) AND NOT #Reset;
	
	#T_notCMD(
	          IN := ( NOT (#sigOffOut OR #sigOnOut) AND #sigFeedBack AND #hasFeedBack AND NOT #Reset),
	          PT := #time_notCMD
	);
	
	#notCMD := (#notCMD OR #T_notCMD.Q) AND NOT #Reset;
	
	
	#wrong_state := (#OnSig AND #OffSig);
	
	//Обобщенная неисправность
	#Fault := #notON OR #notOFF OR #wrong_state OR #notCMD OR #notFeedBack;
	
	IF #DU THEN
	    #setSpeed := #setSpeedDU;
	ELSE
	    #setSpeed := #setSpeedAU;
	END_IF;
	
	
END_FUNCTION_BLOCK

FUNCTION_BLOCK "FB_IM2x3"
{ S7_Optimized_Access := 'FALSE' }
AUTHOR : Aspir
VERSION : 0.1
   VAR_INPUT 
      upSig : Bool;   //       Сигнал верхнего концевика
      midSig : Bool;   //       Сигнал среднего концевика
      dnSig : Bool;   //       Сигнал нижнего концевика
      btnAU : Bool;   // Команда перевода в АУ
      setUp : Bool;   //       Установить в верхнее положение
      setMid : Bool;   //       Установить в среднее положение
      setDn : Bool;   //       Установить в нижнее положение
      Ready : Bool;   //       Условие готовности
      Reset : Bool;   //       Сброс
      btnMU : Bool;   //       Команда на перевод в МУ
      btnMU_ON : Bool;   //       Включить в местном управлении
      btnMU_OF : Bool;   //       Отключить в местном управлении
      sync_sig : Bool;   // сигнал синхронизации
      set_time_notRun : Time;   //       установка времени на не верх
   END_VAR

   VAR_OUTPUT 
      AU : Bool;
      MU : Bool;
      Fault : Bool;   //       Неисправность
      outUp : Bool;   //       Сигнал о движении вверх (вперед)
      outDn : Bool;   //       Сигнал о движении вниз (назад)
      wrong_state : Bool;
      wrong_CMD : Bool;
      notUp : Bool;   //       Сигнал не верх
      notMid : Bool;   //       Сигнал не середина
      notDn : Bool;   //       Сигнал не низ
   END_VAR

   VAR 
      CMD_Up_trig : Bool;
      CMD_Dn_trig : Bool;
      CMD_Dn_MU_trig : Bool;
      CMD_Up_MU_trig : Bool;
      UpState : Bool;
      DnState : Bool;
      MidState : Bool;
      btnMU_ON_old : Bool;
      btnMU_OF_old : Bool;
      syncTask : Bool;
      noRun_timer {InstructionName := 'TON'; LibVersion := '1.0'; S7_SetPoint := 'False'} : TON;
      Antitremble_timer {InstructionName := 'TON'; LibVersion := '1.0'} : TON;
   END_VAR

   VAR_TEMP 
      btnON_front : Bool;
      btnOF_front : Bool;
      move_down : Bool;
      move_up : Bool;
      moving : Bool;
   END_VAR


BEGIN
	IF (#btnAU) THEN
	    #MU := FALSE;
	    #AU := TRUE;
	END_IF;
	
	IF (#btnMU) THEN
	    #MU := TRUE;
	    #AU := FALSE;
	END_IF;
	
	IF (NOT (#AU OR #MU)) THEN
	    #MU := TRUE;
	    #AU := FALSE;
	END_IF;
	
	// триггер фронтов кнопок
	#btnON_front := #btnMU_ON AND NOT #btnMU_ON_old;
	#btnOF_front := #btnMU_OF AND NOT #btnMU_OF_old;
	
	#CMD_Dn_MU_trig := #MU AND ((#CMD_Dn_MU_trig OR #btnOF_front) AND NOT #btnON_front);
	#CMD_Up_MU_trig := #MU AND ((#CMD_Up_MU_trig OR #btnON_front) AND NOT #btnOF_front);
	
	// определение состояний
	IF (#UpState) THEN
	    #CMD_Dn_trig := #AU AND (#CMD_Dn_trig OR (#setMid OR #setDn)) AND NOT #setUp;
	    #CMD_Up_trig := FALSE;
	    
	    IF ((#CMD_Dn_MU_trig OR #CMD_Dn_trig) AND (#midSig OR #dnSig)) THEN
	        #MidState := #midSig;
	        #DnState := #dnSig;
	        #UpState := FALSE;
	        #CMD_Dn_MU_trig := FALSE;
	        #CMD_Dn_trig := FALSE;
	    END_IF;
	    
	ELSIF (#MidState) THEN
	    #CMD_Dn_trig := #AU AND (#CMD_Dn_trig OR #setDn) AND NOT (#setUp OR #setMid);
	    #CMD_Up_trig := #AU AND (#CMD_Up_trig OR #setUp) AND NOT (#setDn OR #setMid);
	    IF ((#CMD_Up_trig OR #CMD_Up_MU_trig) AND #upSig) THEN // едем вверх из среднего
	
	            #UpState := True;
	            #MidState := FALSE;
	            #CMD_Up_trig := FALSE;
	            #CMD_Up_MU_trig := FALSE;
	            
	    END_IF;
	    
	    IF ((#CMD_Dn_MU_trig OR #CMD_Dn_trig) AND #dnSig) THEN
	        
	        #DnState := TRUE;
	        #MidState := FALSE;
	        #CMD_Dn_trig := FALSE;
	        #CMD_Dn_MU_trig := FALSE;
	        
	    END_IF;
	    
	ELSIF (#DnState) THEN
	    #CMD_Up_trig := #AU AND (#CMD_Up_trig OR (#setMid OR #setUp)) AND NOT #setDn;
	    #CMD_Dn_trig := FALSE;
	    
	    IF ((#CMD_Up_trig OR #CMD_Up_MU_trig) AND (#midSig OR #upSig)) THEN // едем по причинам в среднее положение
	            #DnState := FALSE;
	            #MidState := #midSig;
	            #UpState := #upSig;
	            
	            #CMD_Up_trig := FALSE;
	            #CMD_Up_MU_trig := FALSE;
	    END_IF;
	   
	ELSE // инициализация
	    #DnState := TRUE;
	    #MidState := FALSE;
	    #UpState := FALSE;
	END_IF;
	
	#move_down := #CMD_Dn_MU_trig OR #CMD_Dn_trig;
	#move_up := #CMD_Up_MU_trig OR #CMD_Up_trig;
	#moving := #move_up OR #move_down;
	
	// команды гидростанции плюс синхронизация с датчиком
	// 
	#syncTask := (#syncTask OR ((#MidState AND NOT #midSig) OR (#UpState AND NOT #upSig)) AND #sync_sig) AND NOT ((#MidState AND #midSig) OR (#UpState AND #upSig)) AND NOT #moving;
	
	//ошибки
	//
	#noRun_timer(IN:= #AU AND ((#setUp AND NOT #UpState) OR (#setDn AND NOT #dnSig) OR (#setMid AND NOT #MidState)) AND NOT #Reset,
	            PT:=#set_time_notRun);
	#notUp := (#notUp OR (#noRun_timer.Q AND #setUp AND NOT #UpState)) AND NOT #Reset;
	#notDn := (#notDn OR (#noRun_timer.Q AND #setDn AND NOT #dnSig)) AND NOT #Reset;
	#notMid := (#notMid OR (#noRun_timer.Q AND #setMid AND NOT #MidState)) AND NOT #Reset;
	
	(* #noDn_timer(IN:=#AU AND #setDn AND NOT #dnSig AND NOT #Reset,
	            PT:=#set_time_notDn);
	#notDn := (#notDn OR #noDn_timer.Q) AND NOT #Reset;
	
	#noMid_timer(IN:=#AU AND #setMid AND NOT #MidState AND NOT #Reset,
	             PT:=#set_time_notMid);
	#notMid := (#notMid OR #noMid_timer.Q) AND NOT #Reset; *)
	
	#wrong_state := #upSig AND #midSig OR #upSig AND #dnSig OR #midSig AND #dnSig;
	#wrong_CMD := (#wrong_CMD OR (#move_up AND #move_down)) AND NOT #Reset;
	
	#Fault := #wrong_CMD OR #wrong_state OR #notDn OR #notUp OR #notMid;
	
	
	// сигналы клапанам
	#outUp := #Ready AND (#move_up OR #syncTask) AND NOT #upSig AND NOT #Fault;
	#outDn := #Ready AND #move_down AND NOT #dnSig AND NOT #Fault;
	
	// фронты
	// 
	#btnMU_ON_old := #btnMU_ON;
	#btnMU_OF_old := #btnMU_OF;
END_FUNCTION_BLOCK

FUNCTION_BLOCK "FB_HySt_Drive_PassValve"
{ S7_Optimized_Access := 'FALSE' }
VERSION : 0.1
   VAR_INPUT 
      OnSig : Bool;   // сигнал обратной связи двигателя
      Ready : Bool;   // сигнал готовности
      Reset : Bool;   // сброс ошибки
      sigValveFault : Bool;   // сигнал ошибки открытия катушек
      PerepuskOn : Bool;   // сигнал на открытие перепускного клапана
      PumpOn : Bool;   // включение насоса станции
      Set_T_notOn : Time;   // установка времени таймера на невключение
      Set_T_notOFF : Time;   // установка времени таймера на невыключение
   END_VAR

   VAR_OUTPUT 
      CMD_DriveOn : Bool;   // команда включение двигателя
      CMD_PassValveOn : Bool;   // команда открытие перепускного клапана
      Fault : Bool;   // выпал в ошибку
      notOn : Bool;   // ошибка невключения
      notOff : Bool;   // ошибка невыключения
      wrongValveState : Bool;   // ошибка открытия катушек
   END_VAR

   VAR 
      T_notOn_Ton {InstructionName := 'TON'; LibVersion := '1.0'; S7_SetPoint := 'False'} : TON;   // таймер невключения
      T_notOff_Ton {InstructionName := 'TON'; LibVersion := '1.0'; S7_SetPoint := 'False'} : TON;   // таймер невыключения
   END_VAR


BEGIN
	#CMD_DriveOn := #Ready AND #PumpOn AND NOT #Fault;
	
	#CMD_PassValveOn := #Ready AND #PerepuskOn AND NOT #Fault;
	
	#T_notOn_Ton(
	             IN:= #CMD_DriveOn AND NOT #OnSig AND NOT #Reset,
	             PT := #Set_T_notOn
	);
	
	#notOn := (#notOn OR #T_notOn_Ton.Q) AND NOT #Reset;
	
	#T_notOff_Ton(
	              IN := NOT #CMD_DriveOn AND #OnSig AND NOT #Reset,
	              PT := #Set_T_notOFF
	);
	
	#notOff := (#notOff OR #T_notOff_Ton.Q) AND NOT #Reset;
	#wrongValveState := (#wrongValveState OR #sigValveFault) AND NOT #Reset;
	
	
	
	#Fault := #notOff OR #notOn OR #wrongValveState;
	
END_FUNCTION_BLOCK

FUNCTION_BLOCK "FB_IM"
{ S7_Optimized_Access := 'FALSE' }
VERSION : 0.1
// Загрузка
   VAR 
      M_211_Load_Transp : "FB_IM2x1";   //     Загрузочный транспортер пакета
      M_311_Strip_Remov : "FB_IM1x1";   //     Ленточный транспортер удаления рейки
      M_212_Sort_Elevator : "FB_IM2x2S";   //     Загрузочный лифт сортировки+тормоз
      M_213_ConvElevator : "FB_IM1x1";   //     Наклонный транспортер после Лифта
      M_222_Main_Sort_Slide : "FB_IM1x1";   //     Основная горка сортировки Сортировка
      M_325_Tr_Hill : "FB_IM1x1";   //     Транспортер приема доски с Горки перед поштучкой
      M_223_Evaluation_area : "FB_IM1x1";   //     Транспортер после поштучной выдачи(Зона оценки)
      M_224_Individ_dispensing : "FB_IM2x2S";   //     Упоры Поштучной выдачи
      M_225_Conveyor_with_lugs : "FB_IM1x1";   //     Транспортер с бобышками после второй поштучной выдачи
      M_235_Movable_board : "FB_IM2x2S";   //     Подвижный борт
      M_231_Roller_conveyor : "FB_IM1x1";   //     Рольганг Что-то еще
      M_323_Small_Chain : "FB_IM1x1";   // Маленький цепной после элеватора
      M_214_Gasket_receiver : "FB_IM1x1";   // Приемный транспортер прокладок
      M_312_First_slide : "FB_IM1x1";   // Первая горка после приемного транспортера прокладок
      M_313_AF_slide_conv : "FB_IM1x1";   // Транспортер после первой горки прокладок
      M_316_Padloader_IN2 : "FB_IM1x1";   // Транспортер загрузки прокладок в горку 2
      M_314_Second_slide : "FB_IM1x1";   // Вторая горка прокладок
      M_315_Third_slide : "FB_IM1x1";   // Третья горка прокладок
      M_234_Carousel_loader : "FB_IM1x1";   // Транспортер загрузки прокладок перед каруселью
      M_330_Scrap_Conv : "FB_IM1x1";   // Ленточный транспортер брака
      M_331_Scrap_conveyor : "FB_IM1x1";   // Ленточный транспортер приема брака
      M_332_Dump_lug_conv : "FB_IM1x1";   // Транспортер с бобышками сброса с рольганга брака
      M_333_Defective_roller : "FB_IM1x1";   // Рольганг брака после ленточного
      M_334_Layer_set_conv : "FB_IM1x1";   // Транспортер набора слоя брака перед ПФМ
      M_335_Lay_fork_scrap : "FB_IM2x2";   //  M335 Вилы брака ПФМ
      M_336_PFM_elevator : "FB_IM2x2S";   // М336 Лифт брака ПФМ+тормоз
   END_VAR


BEGIN
	
	// --------------------------------------------------ЗАГРУЗКА-------------------------------------------
	//
	REGION Board_loading
	    // Statement section REGION
	    (*
	F211K1_211K2    I       1.0    BOOL    М211 включен сигналы
	E76.7    I      24.7    BOOL    вперед М211 приемный транспортер в автомате
	K1-211X1    Q       1.0    BOOL    М211 вперед загрузочный транспортер
	K1-211X1.1    Q       1.1    BOOL    М211 назад загрузочный транспортер
	S76_2    I      24.2    BOOL    Подтверждение ошибки
	E82_2    I      30.2    BOOL    Приемный транспортер назад ОР2
	S81_1    I      30.1    BOOL    Приемный транспортер вперед ОР2
	
	*)
	    
	    #M_211_Load_Transp(OnSig := "DGI".F211K1_211K2,
	                       //OnCom:=false,,
	                       Ready := "ALG".Ready_loading,
	                       Reset := "DGI".S76_2 OR "ALG".Reset,
	                       btnAU := "ALG".Auto_loading OR "ServDB".M_211.BtnAU,
	                       btnDU := #M_211_Load_Transp.btnDU,
	                       prmDU := TRUE,
	                       btnDU_ON := "ServDB".M_211.BtnFwd,
	                       btnDU_OF := "ServDB".M_211.BtnCmdStop,
	                       btnMU := NOT "ALG".Auto_loading,
	                       btnMU_ON := "DGI".S81_1 OR "DGI".E82_2,
	                       btnMU_OF := "ALG".Auto_loading OR "ServDB".M_211.BtnDU OR NOT ("DGI".S81_1 OR "DGI".E82_2),
	                       btn_Back_ON := "DGI".E82_2 OR "ServDB".M_211.BtnBwd,
	                       btn_Back_OFF := NOT ("DGI".E82_2 OR "ServDB".M_211.BtnBwd),
	                       Set_T_notON := T#500ms,
	                       Set_T_notOFF := T#500ms,
	                       //setSpeedAU := ,
	                       setSpeedDU := "ServDB".M_211.SetSpeedDU,
	                       AU => "ServDB".M_211.AU,
	                       DU => "ServDB".M_211.DU,
	                       MU => "ServDB".M_211.MU,
	                       BACK => "ServDB".M_211.BACK,
	                       Alarm => "ServDB".M_211.Alarm,
	                       Fault => "ServDB".M_211.Fault,
	                       onOutFWD => "ServDB".M_211.CMD_ON,
	                       onOutBWD => "ServDB".M_211.CMD_OFF,
	                       PRM_btnDU_ON => "ServDB".M_211.PrmBtnDU_ON,
	                       PRM_btnDU_OFF => "ServDB".M_211.PrmBtnDU_OF,
	                       PRMbtn_Back_ON => "ServDB".M_211.PRMbtn_Back_ON,
	                       PRMbtn_Back_OFF => "ServDB".M_211.PRMbtn_Back_OFF
	
	    );
	    
	    "K1-211X1" := #M_211_Load_Transp.onOutFWD;
	    "K1-211X1.1" := #M_211_Load_Transp.onOutBWD;
	    
	        
	        
	        (*
	    F311K1_311K2    I       4.0    BOOL    М311 включен сигналы
	    K1_311X1    Q       3.4    BOOL    запуск М311 вперед удаление прокладок ленточный
	    K1_311X1_1    Q       3.5    BOOL    запуск М311 назад удаление прокладок ленточный
	    
	    *)                     
	    #M_311_Strip_Remov(OnSig := "DGI".F311K1_311K2,
	                       Ready := "ALG".Ready_Sorting,
	                       Reset := "DGI".S76_2 OR "ALG".Reset,
	                       btnAU := "ALG".Auto_loading OR "ServDB".M_311.BtnAU,
	                       btnDU := "ServDB".M_311.BtnDU,
	                       prmDU := TRUE,
	                       btnDU_ON := "ServDB".M_311.BtnFwd,
	                       btnDU_OF := "ServDB".M_311.BtnCmdStop,
	                       btnMU := "DGI".E83_1 OR "DGI".E83_2,
	                       btnMU_ON := "DGI".E83_1 OR "DGI".E83_2,
	                       btnMU_OF := NOT ("DGI".E83_1 OR "DGI".E83_2),
	                       Set_T_notON := T#500ms,
	                       Set_T_notOFF := T#500ms,
	                       setSpeedDU := "ServDB".M_311.SetSpeedDU,
	                       AU => "ServDB".M_311.AU,
	                       DU => "ServDB".M_311.DU,
	                       MU => "ServDB".M_311.MU,
	                       Alarm => "ServDB".M_311.Alarm,
	                       Fault => "ServDB".M_311.Fault,
	                       onOutFWD => "ServDB".M_311.CMD_ON,
	                       PRM_btnDU_ON => "ServDB".M_311.PrmBtnDU_ON,
	                       PRM_btnDU_OFF => "ServDB".M_311.PrmBtnDU_OF
	    );
	    
	    "K1-311X1" := #M_311_Strip_Remov.onOutFWD;
	    
	    
	(*
	F212K1    I       1.1    BOOL    Контактор К1 Включен М212 сигналы
	K1-212U    PQW   512    WORD    
	K1_212U2    Q       8.0    BOOL    старт ПЧТ М212
	K1_212U2_2    Q       8.1    BOOL    Реверс ПЧТ М212
	K1-212X1    Q       1.2    BOOL    контактор К1-212 ПЧТ запуск лифт
	K1-212X1.1    Q       1.3    BOOL    Растормаживание М212 лифт
	
	*)
	    #M_212_Sort_Elevator(
	                         onSig := "DGI".Liftdown,
	                         offSig := "DGI".LiftUp,
	                         sigFeedback := "DGI".F212K1 AND "DGI".K1_221U1,
	                         hasFeedback := true,
	                         "Ready" := "ALG".Ready_loading,
	                         Reset := "DGI".S76_2 OR "ALG".Reset,
	                         btnAU := "ServDB".M_212.BtnAU OR "ALG".Auto_loading,
	                         btnDU := "ServDB".M_212.BtnDU,
	                         prmDU := true,
	                         btnUp := "ServDB".M_212.BtnFwd,
	                         btnDown := "ServDB".M_212.BtnBwd,
	                         btnStop := "ServDB".M_212.BtnCmdStop,
	                         btnMU := (*"DGI".S82_4 OR "DGI".E82_5 OR*) NOT ("ServDB".M_212.BtnAU OR "ALG".Auto_loading),
	                         btnMU_ON := "DGI".S82_4,
	                         btnMU_OF := "DGI".E82_5,
	                         set_time_notOn := T#1500ms,
	                         set_time_notOff := T#1500ms,
	                         set_time_notCMD := T#500ms,
	                         setSpeedDU := "ServDB".M_212.SetSpeedDU,
	                         AU => "ServDB".M_212.AU,
	                         DU => "ServDB".M_212.DU,
	                         Fault => "ServDB".M_212.Fault,
	                         outFWD => "ServDB".M_212.CMD_ON,
	                         outBKD => "ServDB".M_212.CMD_OFF
	                         
	    );
	    
	    
	    "K1-212X1" := "ALG".Ready_loading;
	    "K1-212U2" := #M_212_Sort_Elevator.outBKD XOR #M_212_Sort_Elevator.outFWD;
	    "K1-212X1.1" := #M_212_Sort_Elevator.outFWD OR #M_212_Sort_Elevator.outBKD;
	    "K1-212U2.2" := #M_212_Sort_Elevator.outBKD;
	    
	    
	(*
	F213K1    I       1.2    BOOL    контактор К1 Включен М213 сигналы
	K1-213U    PQW   514    WORD    
	K1-213U1    I       7.1    BOOL    ПЧТ 213 в работе сигналы
	K1_213U2    Q       8.2    BOOL    Старт ПЧТ М213
	K1_213X1    Q       1.4    BOOL    контактор К1-213 ПЧТ запуск наклонный транспортер
	
	*)   
	    #M_213_ConvElevator(
	                        OnSig := "DGI".F213K1 AND "DGI".K1_213U1,
	                        Ready := "ALG".Ready_loading OR "ServDB".M_213.Ready,
	                        Reset := "DGI".S76_2 OR "ALG".Reset,
	                        btnAU :=  "ALG".Auto_loading OR "ServDB".M_213.BtnAU,
	                        btnDU := "ServDB".M_213.BtnDU,
	                        prmDU := TRUE,
	                        btnDU_ON := "ServDB".M_213.BtnFwd,
	                        btnDU_OF := NOT "ServDB".M_213.BtnFwd,
	                        btnMU := "DGI".E82_7 OR NOT "DGI".S82_6,
	                        btnMU_ON := "DGI".E82_7,
	                        btnMU_OF := NOT "DGI".E82_7,
	                        Set_T_notON := T#1500ms,
	                        Set_T_notOFF := T#1500ms,
	                        setSpeedDU:= "ServDB".M_213.SetSpeedDU,
	                        AU=> "ServDB".M_213.AU,
	                        DU=>"ServDB".M_213.DU,
	                        MU=>"ServDB".M_213.MU,
	                        Alarm=>"ServDB".M_213.Alarm,
	                        Fault=>"ServDB".M_213.Fault,
	                        onOutFWD=>"ServDB".M_213.CMD_ON,
	                        PRM_btnDU_ON=>"ServDB".M_213.PrmBtnDU_ON,
	                        PRM_btnDU_OFF=> "ServDB".M_213.PrmBtnDU_OF
	    );
	    "K1-213X1" := "ALG".Ready_loading;
	    "K1-213U2" := #M_213_ConvElevator.onOutFWD;
	    
	END_REGION
	
	
	// --------------------------------------------------СОРТИРОВКА-----------------------------------------
	//
	REGION Sorting
	    // Statement section REGION
	    // 
	    
	    
	    (*
	F222K1    I       2.1    BOOL    Контактор К1 Включен М222 сигналы
	K1-222U    PQW   518    WORD    
	K1-222U1    I       7.3    BOOL    ПЧТ 222 в работе сигналы
	K1_222U2    Q       8.5    BOOL    Старт ПЧТ 222
	K1-222X1    Q       2.1    BOOL    Запуск контактора К1-222 ПЧТ маленький цепной после элеватора
	*)
	    
	    #M_222_Main_Sort_Slide(
	                           OnSig := "DGI".F222K1 AND "DGI".K1_222U1,
	                           Ready := "ALG".Ready_Sorting,
	                           Reset := "DGI".S76_2 OR "ALG".Reset,
	                           btnAU := "ServDB".M_222.BtnAU OR "DGI".S77_0,
	                           btnDU := "ServDB".M_222.BtnDU,
	                           prmDU := TRUE,
	                           btnDU_ON := "ServDB".M_222.BtnFwd,
	                           btnDU_OF := "ServDB".M_222.BtnCmdStop,
	                           btnMU := "DGI".E77_1 OR "DGI".E87_2,
	                           btnMU_ON := "DGI".E77_1 OR "DGI".E87_2,
	                           btnMU_OF := NOT ("DGI".E77_1 OR "DGI".E87_2),
	                           Set_T_notON := T#500ms,
	                           Set_T_notOFF := T#500ms,
	                           setSpeedDU := "ServDB".M_222.SetSpeedDU,
	                           AU => "ServDB".M_222.AU,
	                           DU => "ServDB".M_222.DU,
	                           MU => "ServDB".M_222.MU,
	                           Alarm => "ServDB".M_222.Alarm,
	                           Fault => "ServDB".M_222.Fault,
	                           onOutFWD => "ServDB".M_222.CMD_ON,
	                           PRM_btnDU_ON => "ServDB".M_222.PrmBtnDU_ON,
	                           PRM_btnDU_OFF => "ServDB".M_222.PrmBtnDU_OF
	    );
	    
	    "K1-222X1" := "ALG".Ready_Sorting;
	    "K1-222U2" := #M_222_Main_Sort_Slide.onOutFWD;
	    
	    
	    
	    #M_325_Tr_Hill // Транспортер приема доски с Горки перед поштучкой
	(*   
	 F323K1_323K2    I       5.2    BOOL    Резерв
	 K1_325X1    Q       5.2    BOOL    резерв
	 K1_325X1_1    Q       5.3    BOOL    резерв
	 *)
	    (OnSig := #M_325_Tr_Hill.onOutFWD , //"DGI".F325K1 AND "DGI".K1_325U1,
	     Ready := "ALG".Ready_Sorting,
	     Reset := "ALG".Reset OR "DGI".S76_2,
	     btnAU := "ServDB".M_325.BtnAU OR "ALG".Auto_Sorting,
	     btnDU := "ServDB".M_325.BtnDU,
	     prmDU := true,
	     btnDU_ON := "ServDB".M_325.BtnFwd,
	     btnDU_OF := "ServDB".M_325.BtnCmdStop,
	     Set_T_notON := T#500ms,
	     Set_T_notOFF := T#500ms,
	     setSpeedDU := "ServDB".M_325.SetSpeedDU,
	     AU => "ServDB".M_325.AU,
	     DU => "ServDB".M_325.DU,
	     MU => "ServDB".M_325.MU,
	     Alarm => "ServDB".M_325.Alarm,
	     Fault => "ServDB".M_325.Fault,
	     onOutFWD => "ServDB".M_325.CMD_ON,
	     PRM_btnDU_ON => "ServDB".M_325.PrmBtnDU_ON,
	     PRM_btnDU_OFF => "ServDB".M_325.PrmBtnDU_OF,
	     setSpeed => "ServDB".M_325.SetSpeed
	     
	    );
	    
	    "K1-325X1" := "ALG".Ready_Sorting;
	    "K1-325U2" := #M_325_Tr_Hill.onOutFWD;
	    
	    
	    
	    #M_223_Evaluation_area // Транспортер после поштучной выдачи(Зона оценки)
	(*
	F223K1    I       2.2    BOOL    Резерв                            DGI.    F223K1    :=    I       2.2    ; //    Резерв
	K1_223X1    Q       2.2    BOOL    запуск М223 резерва
	*)
	    (OnSig := "DGI".K1_223U1,
	     Ready := "ALG".Ready_Sorting,
	     Reset := "DGI".S76_2 OR "ALG".Reset,
	     btnAU := "ServDB".M_223.BtnAU OR "ALG".Auto_Sorting,
	     btnDU := "ServDB".M_223.BtnDU,
	     prmDU := TRUE,
	     btnDU_ON := "ServDB".M_223.BtnFwd,
	     btnDU_OF := "ServDB".M_223.BtnCmdStop,
	     btnMU :=  "DGI".E76_7 OR NOT "DGI".S76_6,
	     btnMU_ON :="DGI".E76_7,
	     btnMU_OF := NOT "DGI".E76_7,
	     Set_T_notON := T#500ms,
	     Set_T_notOFF := T#500ms,
	     setSpeedDU := "ServDB".M_223.SetSpeedDU,
	     AU => "ServDB".M_223.AU,
	     DU => "ServDB".M_223.DU,
	     MU => "ServDB".M_223.MU,
	     Alarm => "ServDB".M_223.Alarm,
	     Fault => "ServDB".M_223.Fault,
	     onOutFWD => "ServDB".M_223.CMD_ON,
	     PRM_btnDU_ON => "ServDB".M_223.PrmBtnDU_ON,
	     PRM_btnDU_OFF => "ServDB".M_223.PrmBtnDU_OF
	    );
	    
	    "K1-223X1" := "ALG".Ready_Sorting;
	    "K1-223U2" := #M_223_Evaluation_area.onOutFWD;
	    
	    
	    
	    #M_224_Individ_dispensing // Упоры Поштучной выдачи 2x2S
	    (
	     onSig := NOT "DGI".S14_3,
	     offSig:= NOT "DGI".S14_2,
	     sigFeedback:="DGI".F224K1,
	     hasFeedback:=true,
	     btnUp:="ServDB".M_224.BtnFwd,
	     btnDown:="ServDB".M_224.BtnBwd,
	     btnStop:="ServDB".M_224.BtnCmdStop,
	     Ready := "ALG".Ready_Sorting,
	     Reset := "ALG".Reset OR "DGI".S76_2,
	     btnAU := "ALG".Auto_Sorting OR "ServDB".M_224.BtnAU,
	     btnDU := "ServDB".M_224.BtnDU,
	     prmDU := true,
	     
	     btnMU :="DGI".S77_6 OR "DGI".E77_7,
	     btnMU_ON := "DGI".S77_6,
	     btnMU_OF := "DGI".E77_7,
	    
	     set_time_notOn:=T#500ms,
	     set_time_notOff:=T#500ms,
	     set_time_notCMD:=T#500ms,
	     setSpeedDU := "ServDB".M_224.SetSpeedDU,
	     AU => "ServDB".M_224.AU,
	     DU => "ServDB".M_224.DU,
	     MU => "ServDB".M_224.MU,
	    
	     Fault => "ServDB".M_224.Fault,
	     outFWD=> "ServDB".M_224.CMD_ON,
	     outBKD=>"ServDB".M_224.CMD_OFF
	     
	    );
	    
	    "K1-224X1" := #M_224_Individ_dispensing.outFWD;
	    "K1-224-x1.1" := #M_224_Individ_dispensing.outBKD;
	    
	    
	    
	    #M_225_Conveyor_with_lugs // Транспортер с бобышками после второй поштучной выдачи
	(*
	F225K1    I       2.4    BOOL    Контактор К1 Включен М225 сигналы                            DGI.    F225K1    :=    I       2.4    ; //    Контактор К1 Включен М225 сигналы
	K1_225U1    I       7.4    BOOL    Пчт 225 в работе сигналы                            DGI.    K1_225U1    :=    I       7.4    ; //    Пчт 225 в работе сигналы
	B14_0    I      14.0    BOOL    индуктивные датчики 1 М225 (поштучник) кейфазер1                            DGI.    B14_0    :=    I      14.0    ; //    индуктивные датчики 1 М225 (поштучник) кейфазер1
	B14_1    I      14.1    BOOL    индуктивные датчики 2 М225( поштучник) кейфазер2                            DGI.    B14_1    :=    I      14.1    ; //    индуктивные датчики 2 М225( поштучник) кейфазер2
	S14_2    I      14.2    BOOL    Максимальная ширина доски концевик М225 зона                            DGI.    S14_2    :=    I      14.2    ; //    Максимальная ширина доски концевик М225 зона
	S14_3    I      14.3    BOOL    Минимальная ширина доски концевик М225 зона                            DGI.    S14_3    :=    I      14.3    ; //    Минимальная ширина доски концевик М225 зона
	B14_4    I      14.4    BOOL    счет доски М225 зона после бобышек                            DGI.    B14_4    :=    I      14.4    ; //    счет доски М225 зона после бобышек
	B14_5    I      14.5    BOOL    счет доски М225 зона после бобышек                            DGI.    B14_5    :=    I      14.5    ; //    счет доски М225 зона после бобышек
	B14_6    I      14.6    BOOL    счет доски М225 зона после бобышек                            DGI.    B14_6    :=    I      14.6    ; //    счет доски М225 зона после бобышек
	K1_225U    PQW   520    WORD
	K1_225X1    Q       2.5    BOOL    включение контактора К1-225 ПЧТ транспортер бобышек
	K1_225U2    Q       8.6    BOOL    Старт ПЧТ 225
	
	*)
	    (OnSig := "DGI".F225K1 AND "DGI".K1_225U1,
	     Ready := "ALG".Ready_Sorting,
	     Reset := "DGI".S76_2 OR "ALG".Reset,
	     btnAU := "ALG".Auto_Sorting OR "ServDB".M_225.BtnAU,
	     btnDU := "ServDB".M_225.BtnDU,
	     prmDU := TRUE,
	     btnDU_ON := "ServDB".M_225.BtnFwd,
	     btnDU_OF := "ServDB".M_225.BtnCmdStop,
	     Set_T_notON := T#500ms,
	     Set_T_notOFF := T#1s,
	     setSpeedDU := "ServDB".M_225.SetSpeedDU,
	     AU => "ServDB".M_225.AU,
	     DU => "ServDB".M_225.DU,
	     MU => "ServDB".M_225.MU,
	     Alarm => "ServDB".M_225.Alarm,
	     Fault => "ServDB".M_225.Fault,
	     onOutFWD => "ServDB".M_225.CMD_ON,
	     PRM_btnDU_ON => "ServDB".M_225.PrmBtnDU_ON,
	     PRM_btnDU_OFF => "ServDB".M_225.PrmBtnDU_OF
	    );
	    
	    "K1-225X1" := "ALG".Ready_Sorting;
	    "K1-225U2" := #M_225_Conveyor_with_lugs.onOutFWD;
	    
	    
	    
	    #M_235_Movable_board  // Подвижный борт 2x0
	(*
	F235K1_235K2    I       3.4    BOOL    М235 включен сигналы                            DGI.    F235K1_235K2    :=    I       3.4    ; //    М235 включен сигналы
	S80_4    I      28.4    BOOL    поднять, опустить Подвижный борт(М235)                            DGI.    S80_4    :=    I      28.4    ; //    поднять, опустить Подвижный борт(М235)
	S80_5    I      28.5    BOOL    вперед подвижный борт(М235)                            DGI.    S80_5    :=    I      28.5    ; //    вперед подвижный борт(М235)
	E80_6    I      28.6    BOOL    назад подвижный борт(М235)                            DGI.    E80_6    :=    I      28.6    ; //    назад подвижный борт(М235)
	K1_235X1    Q       3.3    BOOL    запуск М235 вперед подвижный борт
	K1_235X1_1    Q       5.7    BOOL    запуск М235 назад подвижный борт
	*)
	    (
	     onSig:="DGI".PodBort_2,
	     offSig:="DGI".PodBort_1,
	     sigFeedback := "DGI".F235K1_235K2,
	     hasFeedback := true,
	     btnUp := "ServDB".M_235.BtnFwd,
	     btnDown := "ServDB".M_235.BtnBwd,
	     btnStop := "ServDB".M_235.BtnCmdStop,
	     Ready := "ALG".Ready_Sorting,
	     Reset := "DGI".S76_2 OR "ALG".Reset,
	     prmDU := TRUE,
	     btnAU := "ServDB".M_235.BtnAU OR "MovableBoard_CTRL_DB".AutoMode,
	     btnDU := "ServDB".M_235.BtnDU AND NOT "MovableBoard_CTRL_DB".AutoMode,
	     btnMU := "DGI".S80_5 OR "DGI".E80_6,
	     btnMU_ON := "DGI".S80_5,
	     btnMU_OF := "DGI".E80_6,
	     set_time_notOn := T#500ms,
	     set_time_notOff := T#500ms,
	     set_time_notCMD := T#500ms,
	     setSpeedDU := "ServDB".M_235.SetSpeedDU,
	     AU => "ServDB".M_235.AU,
	     DU => "ServDB".M_235.DU,
	     MU => "ServDB".M_235.MU,
	     Fault => "ServDB".M_235.Fault,
	     outFWD => "ServDB".M_235.CMD_ON,
	     outBKD => "ServDB".M_235.CMD_OFF
	    );
	    
	    "K1-235X1" := #M_235_Movable_board.outFWD AND "DGI".S76_3;
	    "K1-235X1.1" := #M_235_Movable_board.outBKD AND "DGI".S76_3;
	    
	    
	    #M_231_Roller_conveyor // Рольганг 1x1
	(*
	F231K1    I       3.0    BOOL    Контактор К1 Включен М231 сигналы                            DGI.    F231K1    :=    I       3.0    ; //    Контактор К1 Включен М231 сигналы
	K1_231U1    I       7.5    BOOL    ПЧТ 231 в работе сигналы                            DGI.    K1_231U1    :=    I       7.5    ; //    ПЧТ 231 в работе сигналы
	K1_231U    PQW   522    WORD
	K1_231X1    Q       2.6    BOOL    включение контактора К1-231 ПЧТ ролики торцовочные
	K1_231U2    Q       8.7    BOOL    Старт ПЧТ 231
	
	*)
	    (
	     OnSig := "DGI".F231K1 AND "DGI".K1_231U1,
	     Ready := "ALG".Ready_Sorting,
	     Reset := "DGI".S76_2 OR "ALG".Reset,
	     btnAU := "ALG".Auto_Sorting OR "ServDB".M_213.BtnAU,
	     btnDU := "ServDB".M_213.BtnDU,
	     prmDU := TRUE,
	     btnDU_ON := "ServDB".M_231.BtnFwd,
	     btnDU_OF := "ServDB".M_231.BtnCmdStop,
	     Set_T_notON := T#500ms,
	     Set_T_notOFF := T#500ms,
	     setSpeedDU := "ServDB".M_231.SetSpeedDU,
	     AU => "ServDB".M_231.AU,
	     DU => "ServDB".M_231.DU,
	     MU => "ServDB".M_231.MU,
	     Alarm => "ServDB".M_231.Alarm,
	     Fault => "ServDB".M_231.Fault,
	     onOutFWD => "ServDB".M_231.CMD_ON,
	     PRM_btnDU_ON => "ServDB".M_231.PrmBtnDU_ON,
	     PRM_btnDU_OFF => "ServDB".M_231.PrmBtnDU_OF
	    );
	    
	    "K1-231X1" := "ALG".Ready_Sorting;
	    "K1-231U2" := #M_231_Roller_conveyor.onOutFWD;
	    
	   
	    
	    #M_323_Small_Chain(OnSig := "DGI".F323K1_323K2 AND "DGI".K1_323U1,
	                       Ready := "ALG".Ready_Sorting,
	                       Reset := "DGI".S76_2 OR "ALG".Reset,
	                       btnAU := ("ServDB".M_323.BtnAU OR "ALG".Auto_Sorting),
	                       btnDU:="ServDB".M_323.BtnDU,
	                       prmDU:=true,
	                       btnDU_ON:="ServDB".M_323.BtnFwd,
	                       btnDU_OF:="ServDB".M_323.BtnCmdStop,
	                       (* btnMU :=  "DGI".E76_7 OR NOT "DGI".S76_6,
	                       btnMU_ON :="DGI".E76_7,
	                       btnMU_OF := NOT "DGI".E76_7, *)
	                       Set_T_notON:=T#500ms, 
	                       Set_T_notOFF:=T#500ms,
	                       setSpeedDU:="ServDB".M_323.SetSpeedDU,
	                       AU=>"ServDB".M_323.AU,
	                       DU=>"ServDB".M_323.DU,
	                       MU=>"ServDB".M_323.MU,
	                       Alarm=>"ServDB".M_323.Alarm,
	                       Fault=>"ServDB".M_323.Fault,
	                       onOutFWD=>"ServDB".M_323.CMD_ON,
	                       PRM_btnDU_ON=>"ServDB".M_323.PrmBtnDU_ON,
	                       PRM_btnDU_OFF=>"ServDB".M_323.PrmBtnDU_OF,
	                       setSpeed=>"ServDB".M_323.SetSpeed
	                       
	    );
	    
	    "K1-323X1" := "ALG".Ready_Sorting;
	    "K1-323U2" := #M_323_Small_Chain.onOutFWD;
	    
	END_REGION
	
	
	// ----------------------------------------------Подача прокладок----------------------------------------
	// 
	REGION Gasket_supply
	    // Statement section REGION
	    
	(*
	    М214    Приемный транспортер прокладок (1x1)
	*)
	    #M_214_Gasket_receiver(OnSig:= "DGI".F214K1,
	                           //OnCom:=false,
	                           Ready:= "ALG".Ready_Gasket,
	                           Reset:="DGI".btn_Reset_OP3.ShortTap OR "ALG".Reset,
	                           btnAU:= "ALG".Auto_Gasket OR "ServDB".M_214.BtnAU,
	                           btnDU:= "ServDB".M_214.BtnDU AND NOT "ALG".Auto_Gasket,
	                           prmDU:= TRUE,
	                           btnDU_ON:= "ServDB".M_214.BtnFwd,
	                           btnDU_OF:= NOT "ServDB".M_214.BtnFwd,
	                           //btnMU:="ALG".Auto_Gasket AND NOT "ServDB".M_214.BtnDU,
	                           //btnMU_ON:= "DGI".S214,
	                           //btnMU_OF:= NOT "DGI".S214,
	                           Set_T_notON:=T#500ms,
	                           Set_T_notOFF:=T#500ms,
	                           setSpeedDU:= "ServDB".M_214.SetSpeedDU,
	                           AU=>"ServDB".M_214.AU,
	                           DU=>"ServDB".M_214.DU,
	                           MU=>"ServDB".M_214.MU,
	                           Alarm=> "ServDB".M_214.Alarm,
	                           Fault=>"ServDB".M_214.Fault,
	                           onOutFWD=> "ServDB".M_214.CMD_ON,
	                           PRM_btnDU_ON=> "ServDB".M_214.PrmBtnDU_ON,
	                           PRM_btnDU_OFF=>"ServDB".M_214.PrmBtnDU_OF
	    );
	    
	    "K1-214X1" := #M_214_Gasket_receiver.onOutFWD;
	   
	(*
	         Первая горка после приемного транспортера прокладок
	*)
	    #M_312_First_slide(OnSig:="DGI".F312K1 AND #M_312_First_slide.onOutFWD,// AND "DGI".K1_312U1,
	                       Ready:= "ALG".Ready_Gasket,
	                       Reset:="DGI".btn_Reset_OP3.ShortTap OR "ALG".Reset,
	                       btnAU:= "ALG".Auto_Gasket OR "ServDB".M_312.BtnAU,
	                       btnDU:= "ServDB".M_312.BtnDU AND NOT "ALG".Auto_Gasket,
	                       btnMU := false,
	                       prmDU:= TRUE,
	                       btnDU_ON:= "ServDB".M_312.BtnFwd,
	                       btnDU_OF:= "ServDB".M_312.BtnCmdStop,
	                       Set_T_notON:=T#700ms,
	                       Set_T_notOFF:=T#700ms,
	                       setSpeedDU:= "ServDB".M_312.SetSpeedDU,
	                       AU=>"ServDB".M_312.AU,
	                       DU=>"ServDB".M_312.DU,
	                       MU=>"ServDB".M_312.MU,
	                       Alarm=> "ServDB".M_312.Alarm,
	                       Fault=>"ServDB".M_312.Fault,
	                       onOutFWD=> "ServDB".M_312.CMD_ON,
	                       PRM_btnDU_ON=> "ServDB".M_312.PrmBtnDU_ON,
	                       PRM_btnDU_OFF=>"ServDB".M_312.PrmBtnDU_OF
	    );
	    
	    "K1-312X1" := "ALG".Ready_Gasket;
	    "K1-312U2" :=  #M_312_First_slide.onOutFWD;
	    
	    
	(*
	     М313    Транспортер после первой горки прокладок
	*)
	    #M_313_AF_slide_conv(OnSig:="DGI".F313K1_313K2,
	                         //OnCom:=false,
	                         Ready:= "ALG".Ready_Gasket,
	                         Reset:="DGI".btn_Reset_OP3.ShortTap OR "ALG".Reset,
	                         btnAU:= "ALG".Auto_Gasket OR "ServDB".M_313.BtnAU,
	                         btnDU:= "ServDB".M_313.BtnDU AND NOT "ALG".Auto_Gasket,
	                         prmDU:= TRUE,
	                         btnDU_ON:= "ServDB".M_313.BtnFwd,
	                         btnDU_OF:= "ServDB".M_313.BtnCmdStop,
	                         Set_T_notON:=T#700ms,
	                         Set_T_notOFF:=T#700ms,
	                         setSpeedDU:= "ServDB".M_313.SetSpeedDU,
	                         AU=>"ServDB".M_313.AU,
	                         DU=>"ServDB".M_313.DU,
	                         MU=>"ServDB".M_313.MU,
	                         Alarm=> "ServDB".M_313.Alarm,
	                         Fault=>"ServDB".M_313.Fault,
	                         onOutFWD=> "ServDB".M_313.CMD_ON,
	                         PRM_btnDU_ON=> "ServDB".M_313.PrmBtnDU_ON,
	                         PRM_btnDU_OFF=>"ServDB".M_313.PrmBtnDU_OF
	    );
	    
	    "K1-313X1" := #M_313_AF_slide_conv.onOutFWD;
	    
	    
	(*
	    М316    Транспортер загрузки прокладок в горку 2
	*)
	    #M_316_Padloader_IN2(OnSig:="DGI".F316K1,
	                         //OnCom:=false,
	                         Ready:= "ALG".Ready_Gasket,
	                         Reset:= "DGI".btn_Reset_OP3.ShortTap OR "ALG".Reset,
	                         btnAU:= "ALG".Auto_Gasket OR "ServDB".M_316.BtnAU,
	                         btnDU:= "ServDB".M_316.BtnDU AND NOT "ALG".Auto_Gasket,
	                         prmDU:= TRUE,
	                         btnDU_ON:= "ServDB".M_316.BtnFwd,
	                         btnDU_OF:= NOT "ServDB".M_316.BtnFwd,
	                         Set_T_notON:=T#500ms,
	                         Set_T_notOFF:=T#500ms,
	                         setSpeedDU:= "ServDB".M_316.SetSpeedDU,
	                         AU=>"ServDB".M_316.AU,
	                         DU=>"ServDB".M_316.DU,
	                         MU=>"ServDB".M_316.MU,
	                         Alarm=> "ServDB".M_316.Alarm,
	                         Fault=>"ServDB".M_316.Fault,
	                         onOutFWD=> "ServDB".M_316.CMD_ON,
	                         PRM_btnDU_ON=> "ServDB".M_316.PrmBtnDU_ON,
	                         PRM_btnDU_OFF=>"ServDB".M_316.PrmBtnDU_OF
	    );
	    
	    "K1-316X1" := #M_316_Padloader_IN2.onOutFWD;
	    
	(*
	    М314    Вторая горка прокладок
	*)
	    #M_314_Second_slide(OnSig:="DGI".F314K1,
	                        //OnCom:=false,,
	                        Ready:= "ALG".Ready_Gasket,
	                        Reset:="DGI".btn_Reset_OP3.ShortTap OR "ALG".Reset,
	                        btnAU:="ALG".Auto_Gasket OR "ServDB".M_314.BtnAU,
	                        btnDU:= "ServDB".M_314.BtnDU AND NOT "ALG".Auto_Gasket,
	                        prmDU:= TRUE,
	                        btnDU_ON:= "ServDB".M_314.BtnFwd,
	                        btnDU_OF:= NOT "ServDB".M_314.BtnFwd,
	                        btnMU:= "DGI".E85_4 AND NOT "ServDB".M_314.BtnDU,
	                        btnMU_ON:="DGI".E85_4,
	                        btnMU_OF:= NOT "DGI".E85_4,
	                        Set_T_notON:=T#500ms,
	                        Set_T_notOFF:=T#500ms,
	                        setSpeedDU:= "ServDB".M_314.SetSpeedDU,
	                        AU=>"ServDB".M_314.AU,
	                        DU=>"ServDB".M_314.DU,
	                        MU=>"ServDB".M_314.MU,
	                        Alarm=> "ServDB".M_314.Alarm,
	                        Fault=>"ServDB".M_314.Fault,
	                        onOutFWD=> "ServDB".M_314.CMD_ON,
	                        PRM_btnDU_ON=> "ServDB".M_314.PrmBtnDU_ON,
	                        PRM_btnDU_OFF=>"ServDB".M_314.PrmBtnDU_OF
	    );
	    
	    "K1-314X1" := #M_314_Second_slide.onOutFWD;
	    
	    
	(*
	    М315    Третья горка прокладок
	*)
	    #M_315_Third_slide(OnSig:="DGI".F315K1,
	                       //OnCom:=false,
	                       Ready:= "ALG".Ready_Gasket,
	                       Reset:="DGI".btn_Reset_OP3.ShortTap OR "ALG".Reset,
	                       btnAU:= "ALG".Auto_Gasket OR "ServDB".M_315.BtnAU,
	                       btnDU:= "ServDB".M_315.BtnDU AND NOT "ALG".Auto_Gasket,
	                       prmDU:= TRUE,
	                       btnDU_ON:= "ServDB".M_315.BtnFwd,
	                       btnDU_OF:= NOT "ServDB".M_315.BtnFwd,
	                       btnMU:= "DGI".E85_4,
	                       btnMU_ON:="DGI".E85_4,
	                       btnMU_OF:= NOT "DGI".E85_4,
	                       Set_T_notON:=T#500ms,
	                       Set_T_notOFF:=T#500ms,
	                       setSpeedDU:= "ServDB".M_315.SetSpeedDU,
	                       AU=>"ServDB".M_315.AU,
	                       DU=>"ServDB".M_315.DU,
	                       MU=>"ServDB".M_315.MU,
	                       Alarm=> "ServDB".M_315.Alarm,
	                       Fault=>"ServDB".M_315.Fault,
	                       onOutFWD=> "ServDB".M_315.CMD_ON,
	                       PRM_btnDU_ON=> "ServDB".M_315.PrmBtnDU_ON,
	                       PRM_btnDU_OFF=>"ServDB".M_315.PrmBtnDU_OF
	    );
	    
	    
	    "K1-315X1" := #M_315_Third_slide.onOutFWD;
	    
	(*
	    М234    Транспортер загрузки прокладок перед каруселью
	*)
	    #M_234_Carousel_loader(OnSig:="DGI".F234K1,
	                           Ready:= "ALG".Ready_Gasket,
	                           Reset:="DGI".btn_Reset_OP3.ShortTap OR "ALG".Reset,
	                           btnAU:= "ALG".Auto_Gasket OR "ServDB".M_234.BtnAU,
	                           btnDU:= "ServDB".M_234.BtnDU AND NOT "ALG".Auto_Gasket,
	                           prmDU:= TRUE,
	                           btnDU_ON:= "ServDB".M_234.BtnFwd,
	                           btnDU_OF:= "ServDB".M_234.BtnCmdStop,
	                           btnMU:= "DGI".S85_5 OR "DGI".E85_6,
	                           btnMU_ON:= "DGI".E85_6 OR "DGI".S85_5,
	                           btnMU_OF:= NOT ("DGI".S85_5 OR "DGI".E85_6),
	                           Set_T_notON:=T#1s,
	                           Set_T_notOFF:=T#500ms,
	                           setSpeedDU:= "ServDB".M_234.SetSpeedDU,
	                           AU=>"ServDB".M_234.AU,
	                           DU=>"ServDB".M_234.DU,
	                           MU=>"ServDB".M_234.MU,
	                           Alarm=> "ServDB".M_234.Alarm,
	                           Fault=>"ServDB".M_234.Fault,
	                           onOutFWD=> "ServDB".M_234.CMD_ON,
	                           PRM_btnDU_ON=> "ServDB".M_234.PrmBtnDU_ON,
	                           PRM_btnDU_OFF=>"ServDB".M_234.PrmBtnDU_OF
	                           
	    );
	    
	    "K1-234X1" := #M_234_Carousel_loader.onOutFWD;
	    
	END_REGION
	
	
	// ---------------------------------------------------ПФМ Брака------------------------------------------
	// 
	REGION PFM_Defective
	    // Statement section REGION
	    // 
	    #M_330_Scrap_Conv(OnSig:="DGI".F330K1,
	                      Ready:="ALG".Ready_defect,
	                      Reset:="ALG".Reset OR "DGI".S76_2,
	                      btnAU:= "ALG".Auto_defect OR "ServDB".M_330.BtnAU,
	                      btnDU:="ServDB".M_330.BtnDU,
	                      prmDU:=TRUE,
	                      btnDU_ON:="ServDB".M_330.BtnFwd,
	                      btnDU_OF:="ServDB".M_330.BtnCmdStop,
	                      btnMU := NOT ("ALG".Auto_defect OR "ServDB".M_330.BtnAU),
	                      btnMU_ON := "DGI".S90_1,
	                      btnMU_OF := NOT "DGI".S90_1,
	                      Set_T_notON:=T#500ms,
	                      Set_T_notOFF:=T#500ms,
	                      AU=>"ServDB".M_330.AU,
	                      DU=>"ServDB".M_330.DU,
	                      MU=>"ServDB".M_330.MU,
	                      Alarm=> "ServDB".M_330.Alarm,
	                      Fault=>"ServDB".M_330.Fault,
	                      onOutFWD=>"ServDB".M_330.CMD_ON,
	                      PRM_btnDU_ON=>"ServDB".M_330.PrmBtnDU_ON,
	                      PRM_btnDU_OFF=>"ServDB".M_330.PrmBtnDU_OF);
	    
	    "K1-330X1" := #M_330_Scrap_Conv.onOutFWD;
	    
	    
	    (*
	М331 Ленточный транспортер приема брака (1x1)
	331K1   %I6.0   М331 включен сигналы
	S90.1   %I38.1  М331 вперед ленточный транспортер брака ОР5
	K1-331X1    %Q6.0   запуск М331 ленточный транспортер брака
	*)
	    
	    #M_331_Scrap_conveyor(OnSig := "DGI".F331K1,
	                          //OnCom:= "ПФМ Брака_DB_1".m331.AutoFwd,
	                          Ready := "ALG".Ready_defect,
	                          Reset := "DGI".S76_2,
	                          btnAU := "ALG".Auto_defect OR "ServDB".M_331.BtnAU,
	                          btnDU := "ServDB".M_331.BtnDU,
	                          prmDU := TRUE,
	                          btnDU_ON := "ServDB".M_331.BtnFwd,
	                          btnDU_OF := "ServDB".M_331.BtnCmdStop,
	                          btnMU := NOT ("ALG".Auto_defect OR "ServDB".M_331.BtnAU),
	                          btnMU_ON := "DGI".S90_1,
	                          btnMU_OF := NOT "DGI".S90_1,
	                          Set_T_notON := T#500ms,
	                          Set_T_notOFF := T#500ms,
	                          //setSpeedAU:=0.0,
	                          setSpeedDU := "ServDB".M_331.SetSpeedDU,
	                          AU => "ServDB".M_331.AU,
	                          DU => "ServDB".M_331.DU,
	                          MU => "ServDB".M_331.MU,
	                          Alarm => "ServDB".M_331.Alarm,
	                          Fault => "ServDB".M_331.Fault,
	                          onOutFWD => "ServDB".M_331.CMD_ON,
	                          PRM_btnDU_ON => "ServDB".M_331.PrmBtnDU_ON,
	                          PRM_btnDU_OFF => "ServDB".M_311.PrmBtnDU_OF
	                          //setSpeed => "ServDB".M_311.SetSpeed
	                          
	    );
	    
	    "K1-331X1" := #M_331_Scrap_conveyor.onOutFWD;
	    "ServDB".M_331.ON := "DGI".F331K1;
	    
	(*
	   М332 Транспортер с бобышками сброса с рольганга брака (1x1)
	   K1-332U //no comment
	*)
	    
	    #M_332_Dump_lug_conv(OnSig := "DGI".F332K1 AND "DGI".K1_332U1,
	                         Ready := "ALG".Ready_defect,
	                         Reset := "DGI".S76_2,
	                         btnAU := "ALG".Auto_defect OR "ServDB".M_332.BtnAU,
	                         btnDU := "ServDB".M_332.BtnDU,
	                         prmDU := TRUE,
	                         btnDU_ON := "ServDB".M_332.BtnFwd,
	                         btnDU_OF := "ServDB".M_332.BtnCmdStop,
	                         btnMU := NOT ("ALG".Auto_defect OR "ServDB".M_332.BtnAU),
	                         btnMU_ON := "DGI".S79_4,
	                         btnMU_OF := "DGI".BrakDroper_front,
	                         Set_T_notON := T#500ms,
	                         Set_T_notOFF := T#500ms,
	                         setSpeedDU := "ServDB".M_332.SetSpeedDU,
	                         AU => "ServDB".M_332.AU,
	                         DU => "ServDB".M_332.DU,
	                         MU => "ServDB".M_332.MU,
	                         Alarm => "ServDB".M_332.Alarm,
	                         Fault => "ServDB".M_332.Fault,
	                         onOutFWD => "ServDB".M_332.CMD_ON,
	                         PRM_btnDU_ON => "ServDB".M_332.PrmBtnDU_ON,
	                         PRM_btnDU_OFF => "ServDB".M_332.PrmBtnDU_OF
	    );
	    
	    "K1-332x1" := "ALG".Ready_defect;
	    "K1-332U2" := #M_332_Dump_lug_conv.onOutFWD;
	    
	(*
	    М333 Рольганг брака после ленточного (1x1)
	    K1-333U //no comment
	*)
	    
	    #M_333_Defective_roller(OnSig := "DGI".F333K1 AND "DGI".K1_333U1,
	                            Ready := "ALG".Ready_defect,
	                            Reset := "DGI".S76_2 OR "ALG".Reset,
	                            btnAU := "ALG".Auto_defect OR "ServDB".M_333.BtnAU,
	                            btnDU := "ServDB".M_333.BtnDU,
	                            prmDU := TRUE,
	                            btnDU_ON := "ServDB".M_333.BtnFwd,
	                            btnDU_OF := "ServDB".M_333.BtnCmdStop,
	                            btnMU := NOT ("ALG".Auto_defect OR "ServDB".M_333.BtnAU),
	                            btnMU_ON := "DGI".S90_2,
	                            btnMU_OF := NOT "DGI".S90_2,
	                            Set_T_notON := T#500ms,
	                            Set_T_notOFF := T#500ms,
	                            setSpeedDU := "ServDB".M_333.SetSpeedDU,
	                            AU => "ServDB".M_333.AU,
	                            DU => "ServDB".M_333.DU,
	                            MU => "ServDB".M_333.MU,
	                            Alarm => "ServDB".M_333.Alarm,
	                            Fault =>  "ServDB".M_333.Fault,
	                            onOutFWD => "ServDB".M_333.CMD_ON,
	                            PRM_btnDU_ON => "ServDB".M_333.PrmBtnDU_ON,
	                            PRM_btnDU_OFF => "ServDB".M_333.PrmBtnDU_OF
	    );
	    
	    "K1--333X1" := "ALG".Ready_defect;
	    "K1-333U2" := #M_333_Defective_roller.onOutFWD;
	    
	(*
	    М334 Транспортер набора слоя брака перед ПФМ (1x1)
	    K1-334U // no comment
	*)
	    
	    #M_334_Layer_set_conv(OnSig := "DGI".F334K1 AND "DGI".K1_334U1,
	                          Ready := "ALG".Ready_defect,
	                          Reset := "DGI".S76_2 OR "ALG".Reset,
	                          btnAU := "ALG".Auto_defect OR "ServDB".M_334.BtnAU,
	                          btnDU := "ServDB".M_334.BtnDU AND NOT "ALG".Auto_defect,
	                          prmDU := True,
	                          btnDU_ON := "ServDB".M_334.BtnFwd,
	                          btnDU_OF := "ServDB".M_334.BtnCmdStop,
	                          btnMU := "DGI".S79_5,
	                          btnMU_ON := "DGI".S79_5,
	                          btnMU_OF := NOT "DGI".S79_5,
	                          Set_T_notON := T#500ms,
	                          Set_T_notOFF := T#500ms,
	                         
	                          setSpeedDU := "ServDB".M_334.SetSpeedDU,
	                          AU => "ServDB".M_334.AU,
	                          DU => "ServDB".M_334.DU,
	                          MU => "ServDB".M_334.MU,
	                          Alarm => "ServDB".M_334.Alarm,
	                          Fault => "ServDB".M_334.Fault,
	                          onOutFWD => "ServDB".M_334.CMD_ON,
	                          PRM_btnDU_ON => "ServDB".M_334.PrmBtnDU_ON,
	                          PRM_btnDU_OFF => "ServDB".M_334.PrmBtnDU_OF
	    );
	    
	    "K1-334X1" := "ALG".Ready_defect;
	    "K1-334U2" := #M_334_Layer_set_conv.onOutFWD;
	    
	    
	(* удалить
	"K1-212X1" := "Ready";
	"K1-212U2" := #M_212_Sort_Elevator.outBKD OR #M_212_Sort_Elevator.outFWD;
	"K1-212X1.1" := #M_212_Sort_Elevator.outFWD OR #M_212_Sort_Elevator.outBKD;
	"K1-212U2.2" := #M_212_Sort_Elevator.outBKD;
	*)
	    
	(*
	    M335 Вилы брака ПФМ
	*)
	    
	    #M_335_Lay_fork_scrap(OnSig := "DGI".S22_3,
	                          OffSig := "DGI".S22_2,
	                          sigFeedBack := "DGI".F335K1 AND "DGI".K1_335U1,
	                          hasFeedBack := true,
	                          btnDU_ON := "ServDB".M_335.BtnFwd,
	                          btnDU_OF := "ServDB".M_335.BtnBwd,
	                          Ready := "ALG".Ready_defect,
	                          Reset := "DGI".S76_2 OR "ALG".Reset,
	                          btnAU := "ALG".Auto_defect OR "ServDB".M_335.BtnAU,
	                          btnDU := "ServDB".M_335.BtnDU,
	                          prmDU := TRUE,
	                          btnMU := "DGI".E90_5 OR "DGI".S90_4 OR "DGI".S79_6 OR "DGI".E79_7,
	                          btnMU_ON := "DGI".S90_4 OR "DGI".S79_6,
	                          btnMU_OF :=  "DGI".E90_5 OR "DGI".E79_7,
	                          Set_T_notON := T#17s,
	                          Set_T_notOFF := T#17s,
	                          time_notFeedBack := T#500ms,
	                          time_notCMD := T#500ms,
	                          setSpeedDU := "ServDB".M_335.SetSpeedDU,
	                          AU => "ServDB".M_335.AU,
	                          DU => "ServDB".M_335.DU,
	                          MU => "ServDB".M_335.MU,
	                          Fault => "ServDB".M_335.Fault,
	                          onOutFWD => "ServDB".M_335.CMD_ON,
	                          onOutBWD => "ServDB".M_335.CMD_OFF,
	                          setSpeed=>"ServDB".M_335.SetSpeed
	                          
	    );
	    
	    "K1-335X1" := "ALG".Ready_defect;
	    "K1-335U2" := #M_335_Lay_fork_scrap.onOutBWD OR #M_335_Lay_fork_scrap.onOutFWD;
	    "K1-335U2.2" := #M_335_Lay_fork_scrap.onOutBWD;
	    
	    
	(*
	    М336 Лифт брака ПФМ+тормоз
	*)
	    #M_336_PFM_elevator(onSig := "DGI".B22_5,
	                        offSig := "DGI".B22_4,
	                        sigFeedback := "DGI".F336K1 AND "DGI".K1_336U1,
	                        hasFeedback := TRUE,
	                        btnUp := "ServDB".M_336.BtnFwd,
	                        btnDown := "ServDB".M_336.BtnBwd,
	                        btnStop := "ServDB".M_336.BtnCmdStop,
	                        Ready := "ALG".Ready_defect,
	                        Reset := "DGI".S76_2 OR "ALG".Reset,
	                        prmDU := true,
	                        btnAU := "ALG".Auto_defect OR "ServDB".M_336.BtnAU,
	                        btnDU := "ServDB".M_336.BtnDU,
	                        btnMU := "DGI".E91_1 OR "DGI".S91_0 OR "DGI".S80_2 OR "DGI".E80_3 OR NOT ("ALG".Auto_defect OR "ServDB".M_336.BtnAU OR "ServDB".M_336.BtnDU),
	                        btnMU_ON := "DGI".E91_1 OR "DGI".E80_3 ,
	                        btnMU_OF := "DGI".S91_0 OR "DGI".S80_2,
	                        set_time_notOn := T#500ms,
	                        set_time_notOff := T#500ms,
	                        set_time_notCMD := T#500ms,
	                        setSpeedDU := "ServDB".M_336.SetSpeedDU,
	                        AU => "ServDB".M_336.AU,
	                        DU => "ServDB".M_336.DU,
	                        MU => "ServDB".M_336.MU,
	                        Fault => "ServDB".M_336.Fault,
	                        outFWD => "ServDB".M_336.CMD_ON,
	                        outBKD => "ServDB".M_336.CMD_OFF);
	    
	    
	    "K1-336X1" := "ALG".Ready_defect;
	    "K1-336X1.1" := #M_336_PFM_elevator.outBKD OR #M_336_PFM_elevator.outFWD;
	    "K1-336U2" := #M_336_PFM_elevator.outBKD OR #M_336_PFM_elevator.outFWD;
	    "K1-336U2.2" := #M_336_PFM_elevator.outFWD;
	END_REGION
	
	
	
END_FUNCTION_BLOCK

FUNCTION_BLOCK "FB_IM2x1"
{ S7_Optimized_Access := 'FALSE' }
AUTHOR : Ivanez
VERSION : 0.1
//Абстактный механизм с 1й командой вперед и 1й командой назад, 1й обратной связью (АУ, ДУ)
   VAR_INPUT 
      OnSig : Bool;   //      Сигнал сработавшего состояния
      OnCom : Bool;   //      Команда включения в автоматическом режиме
      Ready : Bool;   //      Условие готовности
      Reset : Bool;   //      Сброс
      btnAU : Bool;   //      Перевести в Автоматическое управление
      btnDU : Bool;   //      Перевести в Дистанционное управление
      prmDU : Bool;   //      Разрешение на перевод в ДУ
      btnDU_ON : Bool;   //      Включить в дистанционном управлении
      btnDU_OF : Bool;   //      Отключить в дистанционном управлении
      btnMU : Bool;   //      Перевести в местное управление
      btnMU_ON : Bool;   //      Включить в местном управлении
      btnMU_OF : Bool;   //      Отключить в местном управлении
      btn_Back_ON : Bool;   //      Включить задний ход
      btn_Back_OFF : Bool;   //      Отключить задний ход
      Set_T_notON : Time;   //      Задержа на формирование невключения
      Set_T_notOFF : Time;   //      Задержа на формирование неотключения
      setSpeedAU : Real;   //      Скорость в режиме автомат
      setSpeedDU : Real;   //      Скорость в режиме ДУoutputs
   END_VAR

   VAR_OUTPUT 
      AU : Bool;   //      Автоматическое управление (АУ)
      DU : Bool;   //      Дистанционное управление (ДУ)
      MU : Bool;   //      Местное управление (ДУ)
      BACK : Bool;   //      Задний ход
      notON : Bool;   //      Предупреждение о невключении
      notOFF : Bool;   //      Предупреждение о неотключении
      Alarm : Bool;   //      Авария (исчезновение готовности при работе)
      Fault : Bool;   //      Неисправность
      onOutFWD : Bool;   //      Сигнал на сработку механизма вперед
      onOutBWD : Bool;   //      Сигнал на сработку механизма назад
      PRM_btnDU_ON : Bool;   //      Разрешение кнопки включения в ДУ
      PRM_btnDU_OFF : Bool;   //      Разрешение кнопки отключения в ДУ
      PRMbtn_Back_ON : Bool;   //      Разрешение кнопки включения заднего хода
      PRMbtn_Back_OFF : Bool;   //      Разрешение кнопки отключения заднего хода
      setSpeed : Real;   //      скорость в автомате для частотникаvariables
   END_VAR

   VAR 
      sigOut : Bool;   //      Сигнал включения
      T_notON_TON {InstructionName := 'TON'; LibVersion := '1.0'; S7_SetPoint := 'False'} : TON;   //      Таймер невключения
      T_notOFF_TON {InstructionName := 'TON'; LibVersion := '1.0'; S7_SetPoint := 'False'} : TON;   //      Таймер неотключения
   END_VAR


BEGIN
	
	//Формирование автоматического управления
	IF #btnAU THEN
	    #AU := true;
	    #DU := false;
	    #MU := false;
	END_IF;
	//Формирование дистанционного управления 
	IF #btnDU THEN
	    #DU := true;
	    #AU := false;
	    #MU := false;
	END_IF;
	//Формирование местного управления
	IF #btnMU THEN
	    #MU := true;
	    #AU := false;
	    #DU := false;
	END_IF;
	
	IF NOT #AU AND NOT #DU AND NOT #MU THEN
	    #MU := true;
	END_IF;
	
	//Разрешения кнопок управления
	#PRM_btnDU_ON := (NOT #OnSig AND #DU OR #notON);
	#PRM_btnDU_OFF := ((#sigOut OR #OnSig) AND #DU OR #notOFF);
	
	//Формирование заднего хода
	#BACK := (#BACK OR #btn_Back_ON AND NOT #OnSig) AND NOT (#btn_Back_OFF AND NOT #OnSig);
	#PRMbtn_Back_ON := NOT #BACK AND NOT #onOutFWD;
	#PRMbtn_Back_OFF := #BACK AND NOT #onOutBWD;
	
	//Формирование выходного сигнала
	#sigOut := #Ready AND ((#sigOut
	OR #AU AND #OnCom
	OR #DU AND #btnDU_ON
	OR #MU AND #btnMU_ON
	)
	AND NOT
	(#Alarm
	OR #AU AND NOT #OnCom
	OR #DU AND #btnDU_OF
	OR #MU AND #btnMU_OF
	OR #notON));
	
	//Выбор выхода ВПЕРЕД НАЗАД
	#onOutBWD := #sigOut AND #BACK;
	#onOutFWD := #sigOut AND NOT #BACK;
	
